LIN {X 0,Y 316.116,Z 363.716,A -85,B 0,C 180,E1 -15587.061,E2 -15587.061} C_VEL
LIN {X 0,Y 317.53,Z 353.599,A -85,B 0,C 180,E1 -15588.551,E2 -15588.551} C_VEL
LIN {X 0,Y 318.947,Z 342.978,A -85,B 0,C 180,E1 -15589.802,E2 -15589.802} C_VEL
LIN {X 0,Y 320.341,Z 331.099,A -85,B 0,C 180,E1 -15590.885,E2 -15590.885} C_VEL
LIN {X 0,Y 321.512,Z 318.732,A -85,B 0,C 180,E1 -15591.729,E2 -15591.729} C_VEL
LIN {X 0,Y 322.42,Z 306.003,A -85,B 0,C 180,E1 -15592.339,E2 -15592.339} C_VEL
LIN {X 0,Y 322.987,Z 292.578,A -85,B 0,C 180,E1 -15592.719,E2 -15592.719} C_VEL
LIN {X 0,Y 324.316,Z 230.091,A -85,B 0,C 180,E1 -15594.097,E2 -15594.097} C_VEL
LIN {X 0,Y 319.347,Z 202.293,A -85,B 0,C 180,E1 -15595.169,E2 -15595.169} C_VEL
LIN {X 0,Y 318.009,Z 197.372,A -85,B 0,C 180,E1 -15595.402,E2 -15595.402} C_VEL
LIN {X 0,Y 316.408,Z 192.985,A -85,B 0,C 180,E1 -15595.706,E2 -15595.706} C_VEL
LIN {X 0,Y 314.523,Z 183.518,A -85,B 0,C 180,E1 -15598.663,E2 -15598.663} C_VEL
LIN {X 0,Y 312.488,Z 174.615,A -85,B 0,C 180,E1 -15601.724,E2 -15601.724} C_VEL
LIN {X 0,Y 312.503,Z 174.545,A -85,B 0,C 180,E1 -15604.209,E2 -15604.209} C_VEL
LIN {X 0,Y 312.511,Z 174.539,A -85,B 0,C 180,E1 -15607.385,E2 -15607.385} C_VEL
LIN {X 0,Y 312.484,Z 174.559,A -85,B 0,C 180,E1 -15610.708,E2 -15610.708} C_VEL
LIN {X 0,Y 312.446,Z 174.564,A -85,B 0,C 180,E1 -15614.209,E2 -15614.209} C_VEL
LIN {X 0,Y 312.478,Z 174.558,A -85,B 0,C 180,E1 -15617.918,E2 -15617.918} C_VEL
LIN {X 0,Y 312.496,Z 174.545,A -85,B 0,C 180,E1 -15620.971,E2 -15620.971} C_VEL
LIN {X 0,Y 312.524,Z 174.52,A -85,B 0,C 180,E1 -15624.219,E2 -15624.219} C_VEL
LIN {X 0,Y 312.496,Z 174.56,A -85,B 0,C 180,E1 -15627.333,E2 -15627.333} C_VEL
LIN {X 0,Y 312.536,Z 174.547,A -85,B 0,C 180,E1 -15631.278,E2 -15631.278} C_VEL
LIN {X 0,Y 312.575,Z 174.542,A -85,B 0,C 180,E1 -15634.71,E2 -15634.71} C_VEL
LIN {X 0,Y 312.524,Z 174.557,A -85,B 0,C 180,E1 -15638.912,E2 -15638.912} C_VEL
LIN {X 0,Y 312.579,Z 174.534,A -85,B 0,C 180,E1 -15641.653,E2 -15641.653} C_VEL
LIN {X 0,Y 312.676,Z 174.535,A -85,B 0,C 180,E1 -15645.685,E2 -15645.685} C_VEL
LIN {X 0,Y 312.693,Z 174.524,A -85,B 0,C 180,E1 -15649.642,E2 -15649.642} C_VEL
LIN {X 0,Y 312.855,Z 174.515,A -85,B 0,C 180,E1 -15652.254,E2 -15652.254} C_VEL
LIN {X 0,Y 312.702,Z 174.515,A -85,B 0,C 180,E1 -15654.842,E2 -15654.842} C_VEL
LIN {X 0,Y 312.979,Z 174.501,A -85,B 0,C 180,E1 -15658.713,E2 -15658.713} C_VEL
LIN {X 0,Y 312.979,Z 174.486,A -85,B 0,C 180,E1 -15661.287,E2 -15661.287} C_VEL
LIN {X 0,Y 312.704,Z 174.531,A -85,B 0,C 180,E1 -15665.158,E2 -15665.158} C_VEL
LIN {X 0,Y 312.862,Z 174.506,A -85,B 0,C 180,E1 -15667.746,E2 -15667.746} C_VEL
LIN {X 0,Y 312.659,Z 174.534,A -85,B 0,C 180,E1 -15671.672,E2 -15671.672} C_VEL
LIN {X 0,Y 312.69,Z 174.521,A -85,B 0,C 180,E1 -15674.888,E2 -15674.888} C_VEL
LIN {X 0,Y 312.621,Z 174.542,A -85,B 0,C 180,E1 -15679.237,E2 -15679.237} C_VEL
LIN {X 0,Y 312.537,Z 174.544,A -85,B 0,C 180,E1 -15682.79,E2 -15682.79} C_VEL
LIN {X 0,Y 312.594,Z 174.546,A -85,B 0,C 180,E1 -15685.936,E2 -15685.936} C_VEL
LIN {X 0,Y 312.537,Z 174.551,A -85,B 0,C 180,E1 -15689.651,E2 -15689.651} C_VEL
LIN {X 0,Y 312.512,Z 174.525,A -85,B 0,C 180,E1 -15693.69,E2 -15693.69} C_VEL
LIN {X 0,Y 312.519,Z 174.539,A -85,B 0,C 180,E1 -15697.386,E2 -15697.386} C_VEL
LIN {X 0,Y 312.484,Z 174.556,A -85,B 0,C 180,E1 -15700.71,E2 -15700.71} C_VEL
LIN {X 0,Y 312.446,Z 174.538,A -85,B 0,C 180,E1 -15704.211,E2 -15704.211} C_VEL
LIN {X 0,Y 312.479,Z 174.555,A -85,B 0,C 180,E1 -15707.92,E2 -15707.92} C_VEL
LIN {X 0,Y 312.494,Z 174.538,A -85,B 0,C 180,E1 -15710.972,E2 -15710.972} C_VEL
LIN {X 0,Y 312.529,Z 174.544,A -85,B 0,C 180,E1 -15714.222,E2 -15714.222} C_VEL
LIN {X 0,Y 312.502,Z 174.56,A -85,B 0,C 180,E1 -15717.335,E2 -15717.335} C_VEL
LIN {X 0,Y 312.588,Z 174.751,A -85,B 0,C 180,E1 -15719.892,E2 -15719.892} C_VEL
LIN {X 0,Y 314.789,Z 184.623,A -85,B 0,C 180,E1 -15723.259,E2 -15723.259} C_VEL
LIN {X 0,Y 315.444,Z 187.959,A -85,B 0,C 180,E1 -15724.271,E2 -15724.271} C_VEL
LIN {X 0,Y 320.254,Z 200.27,A -85,B 0,C 180,E1 -15725.032,E2 -15725.032} C_VEL
LIN {X 0,Y 324.375,Z 221.605,A -85,B 0,C 180,E1 -15725.88,E2 -15725.88} C_VEL
LIN {X 0,Y 322.885,Z 294.83,A -85,B 0,C 180,E1 -15727.527,E2 -15727.527} C_VEL
LIN {X 0,Y 322.027,Z 308.231,A -85,B 0,C 180,E1 -15728.055,E2 -15728.055} C_VEL
LIN {X 0,Y 321.046,Z 321.006,A -85,B 0,C 180,E1 -15728.827,E2 -15728.827} C_VEL
LIN {X 0,Y 319.867,Z 332.351,A -85,B 0,C 180,E1 -15729.755,E2 -15729.755} C_VEL
LIN {X 0,Y 318.375,Z 344.014,A -85,B 0,C 180,E1 -15730.999,E2 -15730.999} C_VEL
LIN {X 0,Y 316.985,Z 354.593,A -85,B 0,C 180,E1 -15732.435,E2 -15732.435} C_VEL
LIN {X 0,Y 315.832,Z 363.045,A -85,B 0,C 180,E1 -15733.851,E2 -15733.851} C_VEL
LIN {X 0,Y 314.535,Z 370.933,A -85,B 0,C 180,E1 -15735.442,E2 -15735.442} C_VEL
LIN {X 0,Y 313.25,Z 378.643,A -85,B 0,C 180,E1 -15737.365,E2 -15737.365} C_VEL
LIN {X 0,Y 312.168,Z 385.722,A -85,B 0,C 180,E1 -15739.625,E2 -15739.625} C_VEL
LIN {X 0,Y 311.5,Z 390.438,A -85,B 0,C 180,E1 -15741.568,E2 -15741.568} C_VEL
LIN {X 0,Y 311.007,Z 394.632,A -85,B 0,C 180,E1 -15743.879,E2 -15743.879} C_VEL
LIN {X 0,Y 310.803,Z 397.316,A -85,B 0,C 180,E1 -15746.111,E2 -15746.111} C_VEL
LIN {X 0,Y 310.698,Z 398.314,A -85,B 0,C 180,E1 -15747.408,E2 -15747.408} C_VEL
LIN {X 0,Y 310.619,Z 399.162,A -85,B 0,C 180,E1 -15750.001,E2 -15750.001} C_VEL
LIN {X 0,Y 310.622,Z 398.969,A -85,B 0,C 180,E1 -15751.297,E2 -15751.297} C_VEL
LIN {X 0,Y 310.697,Z 398.381,A -85,B 0,C 180,E1 -15752.593,E2 -15752.593} C_VEL
LIN {X 0,Y 310.797,Z 397.408,A -85,B 0,C 180,E1 -15753.89,E2 -15753.89} C_VEL
LIN {X 0,Y 311.027,Z 394.734,A -85,B 0,C 180,E1 -15756.157,E2 -15756.157} C_VEL
LIN {X 0,Y 311.497,Z 390.68,A -85,B 0,C 180,E1 -15758.433,E2 -15758.433} C_VEL
LIN {X 0,Y 312.123,Z 386.029,A -85,B 0,C 180,E1 -15760.378,E2 -15760.378} C_VEL
LIN {X 0,Y 313.176,Z 379.019,A -85,B 0,C 180,E1 -15762.639,E2 -15762.639} C_VEL
LIN {X 0,Y 314.476,Z 371.424,A -85,B 0,C 180,E1 -15764.562,E2 -15764.562} C_VEL
LIN {X 0,Y 315.716,Z 363.643,A -85,B 0,C 180,E1 -15766.156,E2 -15766.156} C_VEL
LIN {X 0,Y 317.118,Z 353.168,A -85,B 0,C 180,E1 -15767.894,E2 -15767.894} C_VEL
LIN {X 0,Y 318.634,Z 342.298,A -85,B 0,C 180,E1 -15769.32,E2 -15769.32} C_VEL
LIN {X 0,Y 319.963,Z 331.792,A -85,B 0,C 180,E1 -15770.408,E2 -15770.408} C_VEL
LIN {X 0,Y 321.208,Z 319.141,A -85,B 0,C 180,E1 -15771.415,E2 -15771.415} C_VEL
LIN {X 0,Y 322.223,Z 306.471,A -85,B 0,C 180,E1 -15772.143,E2 -15772.143} C_VEL
LIN {X 0,Y 322.942,Z 294.403,A -85,B 0,C 180,E1 -15772.597,E2 -15772.597} C_VEL
LIN {X 0,Y 324.453,Z 221.803,A -85,B 0,C 180,E1 -15774.224,E2 -15774.224} C_VEL
LIN {X 0,Y 320.487,Z 200.978,A -85,B 0,C 180,E1 -15775.047,E2 -15775.047} C_VEL
LIN {X 0,Y 315.485,Z 188.183,A -85,B 0,C 180,E1 -15775.822,E2 -15775.822} C_VEL
LIN {X 0,Y 314.974,Z 185.72,A -85,B 0,C 180,E1 -15776.504,E2 -15776.504} C_VEL
LIN {X 0,Y 312.776,Z 175.319,A -85,B 0,C 180,E1 -15779.997,E2 -15779.997} C_VEL
LIN {X 0,Y 312.588,Z 174.569,A -85,B 0,C 180,E1 -15780.389,E2 -15780.389} C_VEL
LIN {X 0,Y 312.507,Z 174.544,A -85,B 0,C 180,E1 -15784.21,E2 -15784.21} C_VEL
LIN {X 0,Y 312.521,Z 174.552,A -85,B 0,C 180,E1 -15787.089,E2 -15787.089} C_VEL
LIN {X 0,Y 311.895,Z 174.641,A -85,B 0,C 180,E1 -15788.164,E2 -15788.164} C_VEL
LIN {X 0,Y 309.062,Z 174.996,A -85,B 0,C 180,E1 -15789.915,E2 -15789.915} C_VEL
LIN {X 0,Y 306.618,Z 175.294,A -85,B 0,C 180,E1 -15791.335,E2 -15791.335} C_VEL
LIN {X 0,Y 305.541,Z 175.424,A -85,B 0,C 180,E1 -15792.434,E2 -15792.434} C_VEL
LIN {X 0,Y 305.439,Z 175.436,A -85,B 0,C 180,E1 -15792.807,E2 -15792.807} C_VEL
LIN {X 0,Y 305.454,Z 175.406,A -85,B 0,C 180,E1 -15797.414,E2 -15797.414} C_VEL
LIN {X 0,Y 305.475,Z 175.43,A -85,B 0,C 180,E1 -15801.597,E2 -15801.597} C_VEL
LIN {X 0,Y 305.46,Z 175.388,A -85,B 0,C 180,E1 -15804.886,E2 -15804.886} C_VEL
LIN {X 0,Y 305.45,Z 175.432,A -85,B 0,C 180,E1 -15808.355,E2 -15808.355} C_VEL
LIN {X 0,Y 305.518,Z 175.425,A -85,B 0,C 180,E1 -15811.113,E2 -15811.113} C_VEL
LIN {X 0,Y 305.568,Z 175.42,A -85,B 0,C 180,E1 -15814.087,E2 -15814.087} C_VEL
LIN {X 0,Y 305.477,Z 175.42,A -85,B 0,C 180,E1 -15818.401,E2 -15818.401} C_VEL
LIN {X 0,Y 305.576,Z 175.421,A -85,B 0,C 180,E1 -15821.217,E2 -15821.217} C_VEL
LIN {X 0,Y 305.645,Z 175.399,A -85,B 0,C 180,E1 -15825.349,E2 -15825.349} C_VEL
LIN {X 0,Y 305.634,Z 175.403,A -85,B 0,C 180,E1 -15829.399,E2 -15829.399} C_VEL
LIN {X 0,Y 305.809,Z 175.38,A -85,B 0,C 180,E1 -15832.074,E2 -15832.074} C_VEL
LIN {X 0,Y 305.681,Z 175.405,A -85,B 0,C 180,E1 -15834.723,E2 -15834.723} C_VEL
LIN {X 0,Y 305.952,Z 175.362,A -85,B 0,C 180,E1 -15838.684,E2 -15838.684} C_VEL
LIN {X 0,Y 305.95,Z 175.376,A -85,B 0,C 180,E1 -15841.316,E2 -15841.316} C_VEL
LIN {X 0,Y 305.675,Z 175.391,A -85,B 0,C 180,E1 -15845.277,E2 -15845.277} C_VEL
LIN {X 0,Y 305.767,Z 175.397,A -85,B 0,C 180,E1 -15847.927,E2 -15847.927} C_VEL
LIN {X 0,Y 305.593,Z 175.404,A -85,B 0,C 180,E1 -15851.945,E2 -15851.945} C_VEL
LIN {X 0,Y 305.605,Z 175.418,A -85,B 0,C 180,E1 -15855.014,E2 -15855.014} C_VEL
LIN {X 0,Y 305.543,Z 175.419,A -85,B 0,C 180,E1 -15859.429,E2 -15859.429} C_VEL
LIN {X 0,Y 305.483,Z 175.422,A -85,B 0,C 180,E1 -15863.04,E2 -15863.04} C_VEL
LIN {X 0,Y 305.528,Z 175.426,A -85,B 0,C 180,E1 -15866.221,E2 -15866.221} C_VEL
LIN {X 0,Y 305.485,Z 175.422,A -85,B 0,C 180,E1 -15869.047,E2 -15869.047} C_VEL
LIN {X 0,Y 305.439,Z 175.438,A -85,B 0,C 180,E1 -15871.953,E2 -15871.953} C_VEL
LIN {X 0,Y 305.459,Z 175.406,A -85,B 0,C 180,E1 -15875.114,E2 -15875.114} C_VEL
LIN {X 0,Y 305.447,Z 175.418,A -85,B 0,C 180,E1 -15878.529,E2 -15878.529} C_VEL
LIN {X 0,Y 305.453,Z 175.428,A -85,B 0,C 180,E1 -15882.586,E2 -15882.586} C_VEL
LIN {X 0,Y 305.424,Z 175.436,A -85,B 0,C 180,E1 -15886.345,E2 -15886.345} C_VEL
LIN {X 0,Y 305.456,Z 175.427,A -85,B 0,C 180,E1 -15889.892,E2 -15889.892} C_VEL
LIN {X 0,Y 305.478,Z 175.432,A -85,B 0,C 180,E1 -15893.633,E2 -15893.633} C_VEL
LIN {X 0,Y 305.463,Z 175.515,A -85,B 0,C 180,E1 -15897.759,E2 -15897.759} C_VEL
LIN {X 0,Y 307.544,Z 184.711,A -85,B 0,C 180,E1 -15900.991,E2 -15900.991} C_VEL
LIN {X 0,Y 309.22,Z 192.944,A -85,B 0,C 180,E1 -15903.631,E2 -15903.631} C_VEL
LIN {X 0,Y 312.213,Z 200.76,A -85,B 0,C 180,E1 -15904.151,E2 -15904.151} C_VEL
LIN {X 0,Y 314.705,Z 212.364,A -85,B 0,C 180,E1 -15904.657,E2 -15904.657} C_VEL
LIN {X 0,Y 317.835,Z 230.736,A -85,B 0,C 180,E1 -15905.371,E2 -15905.371} C_VEL
LIN {X 0,Y 316.219,Z 300.948,A -85,B 0,C 180,E1 -15906.982,E2 -15906.982} C_VEL
LIN {X 0,Y 315.294,Z 314.872,A -85,B 0,C 180,E1 -15907.56,E2 -15907.56} C_VEL
LIN {X 0,Y 314.138,Z 327.319,A -85,B 0,C 180,E1 -15908.337,E2 -15908.337} C_VEL
LIN {X 0,Y 312.931,Z 338.417,A -85,B 0,C 180,E1 -15909.285,E2 -15909.285} C_VEL
LIN {X 0,Y 311.387,Z 349.974,A -85,B 0,C 180,E1 -15910.555,E2 -15910.555} C_VEL
LIN {X 0,Y 309.787,Z 360.7,A -85,B 0,C 180,E1 -15912.046,E2 -15912.046} C_VEL
LIN {X 0,Y 308.277,Z 370.627,A -85,B 0,C 180,E1 -15913.798,E2 -15913.798} C_VEL
LIN {X 0,Y 306.817,Z 379.458,A -85,B 0,C 180,E1 -15915.745,E2 -15915.745} C_VEL
LIN {X 0,Y 305.632,Z 386.621,A -85,B 0,C 180,E1 -15917.719,E2 -15917.719} C_VEL
LIN {X 0,Y 304.624,Z 393.142,A -85,B 0,C 180,E1 -15920.035,E2 -15920.035} C_VEL
LIN {X 0,Y 304.056,Z 397.456,A -85,B 0,C 180,E1 -15922.028,E2 -15922.028} C_VEL
LIN {X 0,Y 303.73,Z 401.017,A -85,B 0,C 180,E1 -15924.256,E2 -15924.256} C_VEL
LIN {X 0,Y 303.612,Z 402.976,A -85,B 0,C 180,E1 -15926.017,E2 -15926.017} C_VEL
LIN {X 0,Y 303.585,Z 403.966,A -85,B 0,C 180,E1 -15927.346,E2 -15927.346} C_VEL
LIN {X 0,Y 303.528,Z 404.568,A -85,B 0,C 180,E1 -15928.673,E2 -15928.673} C_VEL
LIN {X 0,Y 303.533,Z 404.78,A -85,B 0,C 180,E1 -15929.999,E2 -15929.999} C_VEL
LIN {X 0,Y 303.585,Z 403.954,A -85,B 0,C 180,E1 -15932.653,E2 -15932.653} C_VEL
LIN {X 0,Y 303.612,Z 402.961,A -85,B 0,C 180,E1 -15933.981,E2 -15933.981} C_VEL
LIN {X 0,Y 303.782,Z 400.858,A -85,B 0,C 180,E1 -15935.841,E2 -15935.841} C_VEL
LIN {X 0,Y 304.094,Z 397.415,A -85,B 0,C 180,E1 -15937.97,E2 -15937.97} C_VEL
LIN {X 0,Y 304.623,Z 393.087,A -85,B 0,C 180,E1 -15939.963,E2 -15939.963} C_VEL
LIN {X 0,Y 305.46,Z 387.573,A -85,B 0,C 180,E1 -15941.95,E2 -15941.95} C_VEL
LIN {X 0,Y 306.61,Z 380.689,A -85,B 0,C 180,E1 -15943.926,E2 -15943.926} C_VEL
LIN {X 0,Y 308.023,Z 372.072,A -85,B 0,C 180,E1 -15945.889,E2 -15945.889} C_VEL
LIN {X 0,Y 309.342,Z 363.431,A -85,B 0,C 180,E1 -15947.484,E2 -15947.484} C_VEL
LIN {X 0,Y 310.813,Z 353.531,A -85,B 0,C 180,E1 -15948.967,E2 -15948.967} C_VEL
LIN {X 0,Y 312.267,Z 342.909,A -85,B 0,C 180,E1 -15950.244,E2 -15950.244} C_VEL
LIN {X 0,Y 313.728,Z 331.028,A -85,B 0,C 180,E1 -15951.346,E2 -15951.346} C_VEL
LIN {X 0,Y 314.943,Z 318.659,A -85,B 0,C 180,E1 -15952.206,E2 -15952.206} C_VEL
LIN {X 0,Y 315.884,Z 305.927,A -85,B 0,C 180,E1 -15952.827,E2 -15952.827} C_VEL
LIN {X 0,Y 316.461,Z 292.492,A -85,B 0,C 180,E1 -15953.215,E2 -15953.215} C_VEL
LIN {X 0,Y 317.799,Z 230.975,A -85,B 0,C 180,E1 -15954.6,E2 -15954.6} C_VEL
LIN {X 0,Y 313.092,Z 204.209,A -85,B 0,C 180,E1 -15955.658,E2 -15955.658} C_VEL
LIN {X 0,Y 311.692,Z 199.331,A -85,B 0,C 180,E1 -15955.903,E2 -15955.903} C_VEL
LIN {X 0,Y 309.197,Z 193.025,A -85,B 0,C 180,E1 -15956.332,E2 -15956.332} C_VEL
LIN {X 0,Y 307.519,Z 184.646,A -85,B 0,C 180,E1 -15959.001,E2 -15959.001} C_VEL
LIN {X 0,Y 305.472,Z 175.62,A -85,B 0,C 180,E1 -15962.142,E2 -15962.142} C_VEL
LIN {X 0,Y 305.458,Z 175.43,A -85,B 0,C 180,E1 -15965.112,E2 -15965.112} C_VEL
LIN {X 0,Y 305.422,Z 175.415,A -85,B 0,C 180,E1 -15968.522,E2 -15968.522} C_VEL
LIN {X 0,Y 305.435,Z 175.437,A -85,B 0,C 180,E1 -15971.856,E2 -15971.856} C_VEL
LIN {X 0,Y 305.394,Z 175.441,A -85,B 0,C 180,E1 -15975.51,E2 -15975.51} C_VEL
LIN {X 0,Y 305.434,Z 175.435,A -85,B 0,C 180,E1 -15978.142,E2 -15978.142} C_VEL
LIN {X 0,Y 305.469,Z 175.41,A -85,B 0,C 180,E1 -15981.596,E2 -15981.596} C_VEL
LIN {X 0,Y 305.455,Z 175.408,A -85,B 0,C 180,E1 -15984.886,E2 -15984.886} C_VEL
LIN {X 0,Y 305.441,Z 175.438,A -85,B 0,C 180,E1 -15988.355,E2 -15988.355} C_VEL
LIN {X 0,Y 305.505,Z 175.421,A -85,B 0,C 180,E1 -15991.112,E2 -15991.112} C_VEL
LIN {X 0,Y 305.562,Z 175.421,A -85,B 0,C 180,E1 -15994.087,E2 -15994.087} C_VEL
LIN {X 0,Y 305.47,Z 175.433,A -85,B 0,C 180,E1 -15998.401,E2 -15998.401} C_VEL
LIN {X 0,Y 305.539,Z 175.412,A -85,B 0,C 180,E1 -16001.214,E2 -16001.214} C_VEL
LIN {X 0,Y 305.616,Z 175.415,A -85,B 0,C 180,E1 -16005.347,E2 -16005.347} C_VEL
LIN {X 0,Y 305.629,Z 175.402,A -85,B 0,C 180,E1 -16009.399,E2 -16009.399} C_VEL
LIN {X 0,Y 305.798,Z 175.393,A -85,B 0,C 180,E1 -16012.074,E2 -16012.074} C_VEL
LIN {X 0,Y 305.674,Z 175.391,A -85,B 0,C 180,E1 -16014.723,E2 -16014.723} C_VEL
LIN {X 0,Y 305.946,Z 175.377,A -85,B 0,C 180,E1 -16018.684,E2 -16018.684} C_VEL
LIN {X 0,Y 305.946,Z 175.362,A -85,B 0,C 180,E1 -16021.316,E2 -16021.316} C_VEL
LIN {X 0,Y 305.84,Z 175.385,A -85,B 0,C 180,E1 -16026.598,E2 -16026.598} C_VEL
LIN {X 0,Y 305.726,Z 175.381,A -85,B 0,C 180,E1 -16029.26,E2 -16029.26} C_VEL
LIN {X 0,Y 305.579,Z 175.417,A -85,B 0,C 180,E1 -16033.297,E2 -16033.297} C_VEL
LIN {X 0,Y 305.584,Z 175.403,A -85,B 0,C 180,E1 -16036.021,E2 -16036.021} C_VEL
LIN {X 0,Y 305.568,Z 175.421,A -85,B 0,C 180,E1 -16039.445,E2 -16039.445} C_VEL
LIN {X 0,Y 305.482,Z 175.425,A -85,B 0,C 180,E1 -16043.042,E2 -16043.042} C_VEL
LIN {X 0,Y 305.524,Z 175.423,A -85,B 0,C 180,E1 -16046.222,E2 -16046.222} C_VEL
LIN {X 0,Y 305.488,Z 175.428,A -85,B 0,C 180,E1 -16049.051,E2 -16049.051} C_VEL
LIN {X 0,Y 305.437,Z 175.431,A -85,B 0,C 180,E1 -16051.953,E2 -16051.953} C_VEL
LIN {X 0,Y 305.455,Z 175.39,A -85,B 0,C 180,E1 -16055.114,E2 -16055.114} C_VEL
LIN {X 0,Y 305.443,Z 175.434,A -85,B 0,C 180,E1 -16058.53,E2 -16058.53} C_VEL
LIN {X 0,Y 305.449,Z 175.409,A -85,B 0,C 180,E1 -16062.587,E2 -16062.587} C_VEL
LIN {X 0,Y 305.421,Z 175.441,A -85,B 0,C 180,E1 -16066.346,E2 -16066.346} C_VEL
LIN {X 0,Y 305.454,Z 175.41,A -85,B 0,C 180,E1 -16069.894,E2 -16069.894} C_VEL
LIN {X 0,Y 305.477,Z 175.429,A -85,B 0,C 180,E1 -16073.633,E2 -16073.633} C_VEL
LIN {X 0,Y 305.462,Z 175.428,A -85,B 0,C 180,E1 -16076.485,E2 -16076.485} C_VEL
LIN {X 0,Y 305.514,Z 175.51,A -85,B 0,C 180,E1 -16079.311,E2 -16079.311} C_VEL
LIN {X 0,Y 307.81,Z 185.73,A -85,B 0,C 180,E1 -16082.931,E2 -16082.931} C_VEL
LIN {X 0,Y 308.278,Z 188.103,A -85,B 0,C 180,E1 -16083.636,E2 -16083.636} C_VEL
LIN {X 0,Y 314.35,Z 203.461,A -85,B 0,C 180,E1 -16084.607,E2 -16084.607} C_VEL
LIN {X 0,Y 317.972,Z 223.57,A -85,B 0,C 180,E1 -16085.408,E2 -16085.408} C_VEL
LIN {X 0,Y 316.28,Z 296.069,A -85,B 0,C 180,E1 -16087.074,E2 -16087.074} C_VEL
LIN {X 0,Y 315.368,Z 309.828,A -85,B 0,C 180,E1 -16087.653,E2 -16087.653} C_VEL
LIN {X 0,Y 314.332,Z 322.174,A -85,B 0,C 180,E1 -16088.438,E2 -16088.438} C_VEL
LIN {X 0,Y 313.007,Z 334.008,A -85,B 0,C 180,E1 -16089.463,E2 -16089.463} C_VEL
LIN {X 0,Y 311.505,Z 345.373,A -85,B 0,C 180,E1 -16090.735,E2 -16090.735} C_VEL
LIN {X 0,Y 310.107,Z 355.391,A -85,B 0,C 180,E1 -16092.149,E2 -16092.149} C_VEL
LIN {X 0,Y 308.726,Z 364.809,A -85,B 0,C 180,E1 -16093.809,E2 -16093.809} C_VEL
LIN {X 0,Y 307.129,Z 373.744,A -85,B 0,C 180,E1 -16095.761,E2 -16095.761} C_VEL
LIN {X 0,Y 305.971,Z 380.937,A -85,B 0,C 180,E1 -16097.734,E2 -16097.734} C_VEL
LIN {X 0,Y 305.159,Z 385.789,A -85,B 0,C 180,E1 -16099.384,E2 -16099.384} C_VEL
LIN {X 0,Y 304.467,Z 390.504,A -85,B 0,C 180,E1 -16101.372,E2 -16101.372} C_VEL
LIN {X 0,Y 304.007,Z 394.113,A -85,B 0,C 180,E1 -16103.363,E2 -16103.363} C_VEL
LIN {X 0,Y 303.819,Z 395.978,A -85,B 0,C 180,E1 -16104.692,E2 -16104.692} C_VEL
LIN {X 0,Y 303.72,Z 397.381,A -85,B 0,C 180,E1 -16106.02,E2 -16106.02} C_VEL
LIN {X 0,Y 303.626,Z 398.38,A -85,B 0,C 180,E1 -16107.347,E2 -16107.347} C_VEL
LIN {X 0,Y 303.535,Z 399.226,A -85,B 0,C 180,E1 -16110.001,E2 -16110.001} C_VEL
LIN {X 0,Y 303.541,Z 399.034,A -85,B 0,C 180,E1 -16111.327,E2 -16111.327} C_VEL
LIN {X 0,Y 303.625,Z 398.445,A -85,B 0,C 180,E1 -16112.654,E2 -16112.654} C_VEL
LIN {X 0,Y 303.714,Z 397.473,A -85,B 0,C 180,E1 -16113.981,E2 -16113.981} C_VEL
LIN {X 0,Y 303.936,Z 395.045,A -85,B 0,C 180,E1 -16116.116,E2 -16116.116} C_VEL
LIN {X 0,Y 304.299,Z 392.029,A -85,B 0,C 180,E1 -16117.966,E2 -16117.966} C_VEL
LIN {X 0,Y 304.861,Z 387.759,A -85,B 0,C 180,E1 -16119.957,E2 -16119.957} C_VEL
LIN {X 0,Y 305.937,Z 381.296,A -85,B 0,C 180,E1 -16122.269,E2 -16122.269} C_VEL
LIN {X 0,Y 307.079,Z 374.196,A -85,B 0,C 180,E1 -16124.243,E2 -16124.243} C_VEL
LIN {X 0,Y 308.644,Z 365.351,A -85,B 0,C 180,E1 -16126.197,E2 -16126.197} C_VEL
LIN {X 0,Y 309.988,Z 355.877,A -85,B 0,C 180,E1 -16127.893,E2 -16127.893} C_VEL
LIN {X 0,Y 311.388,Z 346.231,A -85,B 0,C 180,E1 -16129.274,E2 -16129.274} C_VEL
LIN {X 0,Y 312.943,Z 335.054,A -85,B 0,C 180,E1 -16130.543,E2 -16130.543} C_VEL
LIN {X 0,Y 314.342,Z 322.512,A -85,B 0,C 180,E1 -16131.648,E2 -16131.648} C_VEL
LIN {X 0,Y 315.448,Z 309.573,A -85,B 0,C 180,E1 -16132.472,E2 -16132.472} C_VEL
LIN {X 0,Y 316.29,Z 296.811,A -85,B 0,C 180,E1 -16133.013,E2 -16133.013} C_VEL
LIN {X 0,Y 317.119,Z 265.233,A -85,B 0,C 180,E1 -16133.765,E2 -16133.765} C_VEL
LIN {X 0,Y 317.973,Z 222.627,A -85,B 0,C 180,E1 -16134.731,E2 -16134.731} C_VEL
LIN {X 0,Y 314.219,Z 203.145,A -85,B 0,C 180,E1 -16135.53,E2 -16135.53} C_VEL
LIN {X 0,Y 308.264,Z 188.057,A -85,B 0,C 180,E1 -16136.491,E2 -16136.491} C_VEL
LIN {X 0,Y 306.44,Z 179.396,A -85,B 0,C 180,E1 -16139.366,E2 -16139.366} C_VEL
LIN {X 0,Y 305.509,Z 175.49,A -85,B 0,C 180,E1 -16140.835,E2 -16140.835} C_VEL
LIN {X 0,Y 305.463,Z 175.418,A -85,B 0,C 180,E1 -16145.113,E2 -16145.113} C_VEL
LIN {X 0,Y 305.449,Z 175.424,A -85,B 0,C 180,E1 -16148.528,E2 -16148.528} C_VEL
LIN {X 0,Y 305.454,Z 175.435,A -85,B 0,C 180,E1 -16152.585,E2 -16152.585} C_VEL
LIN {X 0,Y 305.439,Z 175.436,A -85,B 0,C 180,E1 -16152.807,E2 -16152.807} C_VEL
LIN {X 0,Y 304.725,Z 175.526,A -85,B 0,C 180,E1 -16153.907,E2 -16153.907} C_VEL
LIN {X 0,Y 301.828,Z 175.865,A -85,B 0,C 180,E1 -16155.696,E2 -16155.696} C_VEL
LIN {X 0,Y 299.424,Z 176.157,A -85,B 0,C 180,E1 -16157.148,E2 -16157.148} C_VEL
LIN {X 0,Y 298.436,Z 176.289,A -85,B 0,C 180,E1 -16158.273,E2 -16158.273} C_VEL
LIN {X 0,Y 298.378,Z 176.302,A -85,B 0,C 180,E1 -16158.654,E2 -16158.654} C_VEL
LIN {X 0,Y 298.412,Z 176.302,A -85,B 0,C 180,E1 -16162.241,E2 -16162.241} C_VEL
LIN {X 0,Y 298.406,Z 176.268,A -85,B 0,C 180,E1 -16165.581,E2 -16165.581} C_VEL
LIN {X 0,Y 298.393,Z 176.314,A -85,B 0,C 180,E1 -16168.791,E2 -16168.791} C_VEL
LIN {X 0,Y 298.46,Z 176.296,A -85,B 0,C 180,E1 -16171.904,E2 -16171.904} C_VEL
LIN {X 0,Y 298.481,Z 176.304,A -85,B 0,C 180,E1 -16174.923,E2 -16174.923} C_VEL
LIN {X 0,Y 298.433,Z 176.302,A -85,B 0,C 180,E1 -16179.314,E2 -16179.314} C_VEL
LIN {X 0,Y 298.531,Z 176.294,A -85,B 0,C 180,E1 -16182.179,E2 -16182.179} C_VEL
LIN {X 0,Y 298.59,Z 176.276,A -85,B 0,C 180,E1 -16184.994,E2 -16184.994} C_VEL
LIN {X 0,Y 298.59,Z 176.284,A -85,B 0,C 180,E1 -16189.146,E2 -16189.146} C_VEL
LIN {X 0,Y 298.755,Z 176.256,A -85,B 0,C 180,E1 -16191.886,E2 -16191.886} C_VEL
LIN {X 0,Y 298.652,Z 176.281,A -85,B 0,C 180,E1 -16194.599,E2 -16194.599} C_VEL
LIN {X 0,Y 298.918,Z 176.238,A -85,B 0,C 180,E1 -16198.653,E2 -16198.653} C_VEL
LIN {X 0,Y 298.917,Z 176.252,A -85,B 0,C 180,E1 -16201.347,E2 -16201.347} C_VEL
LIN {X 0,Y 298.77,Z 176.263,A -85,B 0,C 180,E1 -16206.754,E2 -16206.754} C_VEL
LIN {X 0,Y 298.621,Z 176.281,A -85,B 0,C 180,E1 -16209.482,E2 -16209.482} C_VEL
LIN {X 0,Y 298.54,Z 176.295,A -85,B 0,C 180,E1 -16213.616,E2 -16213.616} C_VEL
LIN {X 0,Y 298.483,Z 176.299,A -85,B 0,C 180,E1 -16216.412,E2 -16216.412} C_VEL
LIN {X 0,Y 298.483,Z 176.301,A -85,B 0,C 180,E1 -16219.641,E2 -16219.641} C_VEL
LIN {X 0,Y 298.426,Z 176.297,A -85,B 0,C 180,E1 -16223.6,E2 -16223.6} C_VEL
LIN {X 0,Y 298.484,Z 176.304,A -85,B 0,C 180,E1 -16226.575,E2 -16226.575} C_VEL
LIN {X 0,Y 298.414,Z 176.303,A -85,B 0,C 180,E1 -16229.642,E2 -16229.642} C_VEL
LIN {X 0,Y 298.392,Z 176.315,A -85,B 0,C 180,E1 -16232.801,E2 -16232.801} C_VEL
LIN {X 0,Y 298.444,Z 176.267,A -85,B 0,C 180,E1 -16236.808,E2 -16236.808} C_VEL
LIN {X 0,Y 298.385,Z 176.317,A -85,B 0,C 180,E1 -16241.088,E2 -16241.088} C_VEL
LIN {X 0,Y 298.398,Z 176.305,A -85,B 0,C 180,E1 -16243.104,E2 -16243.104} C_VEL
LIN {X 0,Y 298.402,Z 176.307,A -85,B 0,C 180,E1 -16246.921,E2 -16246.921} C_VEL
LIN {X 0,Y 298.389,Z 176.293,A -85,B 0,C 180,E1 -16251.01,E2 -16251.01} C_VEL
LIN {X 0,Y 298.417,Z 176.315,A -85,B 0,C 180,E1 -16253.93,E2 -16253.93} C_VEL
LIN {X 0,Y 298.463,Z 176.375,A -85,B 0,C 180,E1 -16257.208,E2 -16257.208} C_VEL
LIN {X 0,Y 300.544,Z 185.697,A -85,B 0,C 180,E1 -16260.589,E2 -16260.589} C_VEL
LIN {X 0,Y 302.053,Z 192.974,A -85,B 0,C 180,E1 -16262.968,E2 -16262.968} C_VEL
LIN {X 0,Y 306.642,Z 205.052,A -85,B 0,C 180,E1 -16263.756,E2 -16263.756} C_VEL
LIN {X 0,Y 311.027,Z 229.598,A -85,B 0,C 180,E1 -16264.768,E2 -16264.768} C_VEL
LIN {X 0,Y 311.41,Z 233.755,A -85,B 0,C 180,E1 -16264.905,E2 -16264.905} C_VEL
LIN {X 0,Y 309.706,Z 300.897,A -85,B 0,C 180,E1 -16266.469,E2 -16266.469} C_VEL
LIN {X 0,Y 308.76,Z 314.816,A -85,B 0,C 180,E1 -16267.058,E2 -16267.058} C_VEL
LIN {X 0,Y 307.537,Z 327.26,A -85,B 0,C 180,E1 -16267.848,E2 -16267.848} C_VEL
LIN {X 0,Y 306.287,Z 338.356,A -85,B 0,C 180,E1 -16268.814,E2 -16268.814} C_VEL
LIN {X 0,Y 304.698,Z 349.913,A -85,B 0,C 180,E1 -16270.11,E2 -16270.11} C_VEL
LIN {X 0,Y 303.06,Z 360.317,A -85,B 0,C 180,E1 -16271.581,E2 -16271.581} C_VEL
LIN {X 0,Y 301.668,Z 369.306,A -85,B 0,C 180,E1 -16273.166,E2 -16273.166} C_VEL
LIN {X 0,Y 300.199,Z 378.04,A -85,B 0,C 180,E1 -16275.077,E2 -16275.077} C_VEL
LIN {X 0,Y 298.837,Z 385.445,A -85,B 0,C 180,E1 -16277.09,E2 -16277.09} C_VEL
LIN {X 0,Y 297.864,Z 391.391,A -85,B 0,C 180,E1 -16279.119,E2 -16279.119} C_VEL
LIN {X 0,Y 297.199,Z 396.088,A -85,B 0,C 180,E1 -16281.158,E2 -16281.158} C_VEL
LIN {X 0,Y 296.762,Z 399.675,A -85,B 0,C 180,E1 -16283.199,E2 -16283.199} C_VEL
LIN {X 0,Y 296.601,Z 401.525,A -85,B 0,C 180,E1 -16284.561,E2 -16284.561} C_VEL
LIN {X 0,Y 296.516,Z 402.911,A -85,B 0,C 180,E1 -16285.922,E2 -16285.922} C_VEL
LIN {X 0,Y 296.491,Z 403.901,A -85,B 0,C 180,E1 -16287.282,E2 -16287.282} C_VEL
LIN {X 0,Y 296.45,Z 404.504,A -85,B 0,C 180,E1 -16288.641,E2 -16288.641} C_VEL
LIN {X 0,Y 296.451,Z 404.716,A -85,B 0,C 180,E1 -16289.999,E2 -16289.999} C_VEL
LIN {X 0,Y 296.45,Z 404.496,A -85,B 0,C 180,E1 -16291.358,E2 -16291.358} C_VEL
LIN {X 0,Y 296.491,Z 403.889,A -85,B 0,C 180,E1 -16292.717,E2 -16292.717} C_VEL
LIN {X 0,Y 296.64,Z 401.501,A -85,B 0,C 180,E1 -16295.437,E2 -16295.437} C_VEL
LIN {X 0,Y 296.897,Z 398.573,A -85,B 0,C 180,E1 -16297.48,E2 -16297.48} C_VEL
LIN {X 0,Y 297.384,Z 394.61,A -85,B 0,C 180,E1 -16299.521,E2 -16299.521} C_VEL
LIN {X 0,Y 298.356,Z 388.515,A -85,B 0,C 180,E1 -16301.894,E2 -16301.894} C_VEL
LIN {X 0,Y 299.465,Z 381.855,A -85,B 0,C 180,E1 -16303.918,E2 -16303.918} C_VEL
LIN {X 0,Y 300.938,Z 373.592,A -85,B 0,C 180,E1 -16305.926,E2 -16305.926} C_VEL
LIN {X 0,Y 302.285,Z 365.114,A -85,B 0,C 180,E1 -16307.591,E2 -16307.591} C_VEL
LIN {X 0,Y 303.713,Z 355.811,A -85,B 0,C 180,E1 -16309.077,E2 -16309.077} C_VEL
LIN {X 0,Y 305.398,Z 344.267,A -85,B 0,C 180,E1 -16310.544,E2 -16310.544} C_VEL
LIN {X 0,Y 306.909,Z 332.892,A -85,B 0,C 180,E1 -16311.668,E2 -16311.668} C_VEL
LIN {X 0,Y 308.171,Z 321.188,A -85,B 0,C 180,E1 -16312.544,E2 -16312.544} C_VEL
LIN {X 0,Y 309.226,Z 307.689,A -85,B 0,C 180,E1 -16313.258,E2 -16313.258} C_VEL
LIN {X 0,Y 309.908,Z 294.195,A -85,B 0,C 180,E1 -16313.691,E2 -16313.691} C_VEL
LIN {X 0,Y 311.288,Z 231.479,A -85,B 0,C 180,E1 -16315.135,E2 -16315.135} C_VEL
LIN {X 0,Y 306.724,Z 205.539,A -85,B 0,C 180,E1 -16316.195,E2 -16316.195} C_VEL
LIN {X 0,Y 304.353,Z 198.944,A -85,B 0,C 180,E1 -16316.584,E2 -16316.584} C_VEL
LIN {X 0,Y 302.015,Z 193.032,A -85,B 0,C 180,E1 -16316.998,E2 -16316.998} C_VEL
LIN {X 0,Y 301.27,Z 189.184,A -85,B 0,C 180,E1 -16318.188,E2 -16318.188} C_VEL
LIN {X 0,Y 299.079,Z 179.364,A -85,B 0,C 180,E1 -16321.606,E2 -16321.606} C_VEL
LIN {X 0,Y 298.425,Z 176.335,A -85,B 0,C 180,E1 -16322.795,E2 -16322.795} C_VEL
LIN {X 0,Y 298.438,Z 176.299,A -85,B 0,C 180,E1 -16326.805,E2 -16326.805} C_VEL
LIN {X 0,Y 298.382,Z 176.319,A -85,B 0,C 180,E1 -16331.086,E2 -16331.086} C_VEL
LIN {X 0,Y 298.394,Z 176.309,A -85,B 0,C 180,E1 -16333.102,E2 -16333.102} C_VEL
LIN {X 0,Y 298.397,Z 176.305,A -85,B 0,C 180,E1 -16336.92,E2 -16336.92} C_VEL
LIN {X 0,Y 298.397,Z 176.299,A -85,B 0,C 180,E1 -16341.005,E2 -16341.005} C_VEL
LIN {X 0,Y 298.411,Z 176.273,A -85,B 0,C 180,E1 -16343.929,E2 -16343.929} C_VEL
LIN {X 0,Y 298.386,Z 176.316,A -85,B 0,C 180,E1 -16347.983,E2 -16347.983} C_VEL
LIN {X 0,Y 298.45,Z 176.305,A -85,B 0,C 180,E1 -16351.903,E2 -16351.903} C_VEL
LIN {X 0,Y 298.475,Z 176.296,A -85,B 0,C 180,E1 -16354.923,E2 -16354.923} C_VEL
LIN {X 0,Y 298.423,Z 176.311,A -85,B 0,C 180,E1 -16359.313,E2 -16359.313} C_VEL
LIN {X 0,Y 298.496,Z 176.286,A -85,B 0,C 180,E1 -16362.177,E2 -16362.177} C_VEL
LIN {X 0,Y 298.577,Z 176.294,A -85,B 0,C 180,E1 -16364.994,E2 -16364.994} C_VEL
LIN {X 0,Y 298.585,Z 176.277,A -85,B 0,C 180,E1 -16369.146,E2 -16369.146} C_VEL
LIN {X 0,Y 298.744,Z 176.271,A -85,B 0,C 180,E1 -16371.886,E2 -16371.886} C_VEL
LIN {X 0,Y 298.645,Z 176.267,A -85,B 0,C 180,E1 -16374.599,E2 -16374.599} C_VEL
LIN {X 0,Y 298.912,Z 176.253,A -85,B 0,C 180,E1 -16378.653,E2 -16378.653} C_VEL
LIN {X 0,Y 298.912,Z 176.238,A -85,B 0,C 180,E1 -16381.347,E2 -16381.347} C_VEL
LIN {X 0,Y 298.786,Z 176.262,A -85,B 0,C 180,E1 -16386.754,E2 -16386.754} C_VEL
LIN {X 0,Y 298.671,Z 176.26,A -85,B 0,C 180,E1 -16389.481,E2 -16389.481} C_VEL
LIN {X 0,Y 298.542,Z 176.294,A -85,B 0,C 180,E1 -16393.616,E2 -16393.616} C_VEL
LIN {X 0,Y 298.539,Z 176.282,A -85,B 0,C 180,E1 -16396.409,E2 -16396.409} C_VEL
LIN {X 0,Y 298.503,Z 176.302,A -85,B 0,C 180,E1 -16399.655,E2 -16399.655} C_VEL
LIN {X 0,Y 298.449,Z 176.302,A -85,B 0,C 180,E1 -16403.599,E2 -16403.599} C_VEL
LIN {X 0,Y 298.479,Z 176.297,A -85,B 0,C 180,E1 -16406.576,E2 -16406.576} C_VEL
LIN {X 0,Y 298.413,Z 176.31,A -85,B 0,C 180,E1 -16409.642,E2 -16409.642} C_VEL
LIN {X 0,Y 298.388,Z 176.301,A -85,B 0,C 180,E1 -16412.801,E2 -16412.801} C_VEL
LIN {X 0,Y 298.44,Z 176.277,A -85,B 0,C 180,E1 -16416.809,E2 -16416.809} C_VEL
LIN {X 0,Y 298.382,Z 176.31,A -85,B 0,C 180,E1 -16421.089,E2 -16421.089} C_VEL
LIN {X 0,Y 298.394,Z 176.284,A -85,B 0,C 180,E1 -16423.105,E2 -16423.105} C_VEL
LIN {X 0,Y 298.398,Z 176.315,A -85,B 0,C 180,E1 -16426.922,E2 -16426.922} C_VEL
LIN {X 0,Y 298.395,Z 176.293,A -85,B 0,C 180,E1 -16431.009,E2 -16431.009} C_VEL
LIN {X 0,Y 298.415,Z 176.305,A -85,B 0,C 180,E1 -16433.931,E2 -16433.931} C_VEL
LIN {X 0,Y 298.393,Z 176.309,A -85,B 0,C 180,E1 -16437.985,E2 -16437.985} C_VEL
LIN {X 0,Y 298.443,Z 176.418,A -85,B 0,C 180,E1 -16438.798,E2 -16438.798} C_VEL
LIN {X 0,Y 300.538,Z 185.486,A -85,B 0,C 180,E1 -16442.117,E2 -16442.117} C_VEL
LIN {X 0,Y 301.14,Z 188.189,A -85,B 0,C 180,E1 -16442.961,E2 -16442.961} C_VEL
LIN {X 0,Y 308.111,Z 205.736,A -85,B 0,C 180,E1 -16444.11,E2 -16444.11} C_VEL
LIN {X 0,Y 311.52,Z 223.82,A -85,B 0,C 180,E1 -16444.868,E2 -16444.868} C_VEL
LIN {X 0,Y 309.768,Z 296.149,A -85,B 0,C 180,E1 -16446.564,E2 -16446.564} C_VEL
LIN {X 0,Y 308.808,Z 309.904,A -85,B 0,C 180,E1 -16447.151,E2 -16447.151} C_VEL
LIN {X 0,Y 307.763,Z 322.246,A -85,B 0,C 180,E1 -16447.954,E2 -16447.954} C_VEL
LIN {X 0,Y 306.375,Z 334.078,A -85,B 0,C 180,E1 -16448.998,E2 -16448.998} C_VEL
LIN {X 0,Y 304.802,Z 345.442,A -85,B 0,C 180,E1 -16450.294,E2 -16450.294} C_VEL
LIN {X 0,Y 303.4,Z 355.083,A -85,B 0,C 180,E1 -16451.678,E2 -16451.678} C_VEL
LIN {X 0,Y 301.907,Z 364.877,A -85,B 0,C 180,E1 -16453.432,E2 -16453.432} C_VEL
LIN {X 0,Y 300.25,Z 373.811,A -85,B 0,C 180,E1 -16455.427,E2 -16455.427} C_VEL
LIN {X 0,Y 299.025,Z 381.004,A -85,B 0,C 180,E1 -16457.444,E2 -16457.444} C_VEL
LIN {X 0,Y 298.168,Z 385.855,A -85,B 0,C 180,E1 -16459.132,E2 -16459.132} C_VEL
LIN {X 0,Y 297.424,Z 390.57,A -85,B 0,C 180,E1 -16461.166,E2 -16461.166} C_VEL
LIN {X 0,Y 296.947,Z 394.179,A -85,B 0,C 180,E1 -16463.205,E2 -16463.205} C_VEL
LIN {X 0,Y 296.748,Z 396.044,A -85,B 0,C 180,E1 -16464.565,E2 -16464.565} C_VEL
LIN {X 0,Y 296.64,Z 397.447,A -85,B 0,C 180,E1 -16465.925,E2 -16465.925} C_VEL
LIN {X 0,Y 296.555,Z 398.445,A -85,B 0,C 180,E1 -16467.284,E2 -16467.284} C_VEL
LIN {X 0,Y 296.454,Z 399.291,A -85,B 0,C 180,E1 -16470.001,E2 -16470.001} C_VEL
LIN {X 0,Y 296.463,Z 399.099,A -85,B 0,C 180,E1 -16471.359,E2 -16471.359} C_VEL
LIN {X 0,Y 296.554,Z 398.509,A -85,B 0,C 180,E1 -16472.717,E2 -16472.717} C_VEL
LIN {X 0,Y 296.634,Z 397.537,A -85,B 0,C 180,E1 -16474.076,E2 -16474.076} C_VEL
LIN {X 0,Y 296.83,Z 395.39,A -85,B 0,C 180,E1 -16476.048,E2 -16476.048} C_VEL
LIN {X 0,Y 297.269,Z 392.093,A -85,B 0,C 180,E1 -16478.155,E2 -16478.155} C_VEL
LIN {X 0,Y 297.855,Z 387.823,A -85,B 0,C 180,E1 -16480.193,E2 -16480.193} C_VEL
LIN {X 0,Y 298.983,Z 381.36,A -85,B 0,C 180,E1 -16482.559,E2 -16482.559} C_VEL
LIN {X 0,Y 300.199,Z 374.259,A -85,B 0,C 180,E1 -16484.577,E2 -16484.577} C_VEL
LIN {X 0,Y 301.809,Z 365.414,A -85,B 0,C 180,E1 -16486.574,E2 -16486.574} C_VEL
LIN {X 0,Y 303.178,Z 356.247,A -85,B 0,C 180,E1 -16488.254,E2 -16488.254} C_VEL
LIN {X 0,Y 304.703,Z 346.291,A -85,B 0,C 180,E1 -16489.714,E2 -16489.714} C_VEL
LIN {X 0,Y 306.321,Z 335.114,A -85,B 0,C 180,E1 -16491.007,E2 -16491.007} C_VEL
LIN {X 0,Y 307.742,Z 322.57,A -85,B 0,C 180,E1 -16492.137,E2 -16492.137} C_VEL
LIN {X 0,Y 308.911,Z 309.627,A -85,B 0,C 180,E1 -16492.974,E2 -16492.974} C_VEL
LIN {X 0,Y 309.783,Z 296.86,A -85,B 0,C 180,E1 -16493.525,E2 -16493.525} C_VEL
LIN {X 0,Y 310.631,Z 265.902,A -85,B 0,C 180,E1 -16494.277,E2 -16494.277} C_VEL
LIN {X 0,Y 311.48,Z 223.339,A -85,B 0,C 180,E1 -16495.265,E2 -16495.265} C_VEL
LIN {X 0,Y 308.148,Z 205.778,A -85,B 0,C 180,E1 -16496.004,E2 -16496.004} C_VEL
LIN {X 0,Y 301.137,Z 188.253,A -85,B 0,C 180,E1 -16497.155,E2 -16497.155} C_VEL
LIN {X 0,Y 300.359,Z 184.699,A -85,B 0,C 180,E1 -16498.283,E2 -16498.283} C_VEL
LIN {X 0,Y 298.503,Z 176.636,A -85,B 0,C 180,E1 -16501.196,E2 -16501.196} C_VEL
LIN {X 0,Y 298.415,Z 176.303,A -85,B 0,C 180,E1 -16501.782,E2 -16501.782} C_VEL
LIN {X 0,Y 298.432,Z 176.3,A -85,B 0,C 180,E1 -16506.068,E2 -16506.068} C_VEL
LIN {X 0,Y 298.403,Z 176.289,A -85,B 0,C 180,E1 -16509.487,E2 -16509.487} C_VEL
LIN {X 0,Y 298.398,Z 176.315,A -85,B 0,C 180,E1 -16513.103,E2 -16513.103} C_VEL
LIN {X 0,Y 298.402,Z 176.282,A -85,B 0,C 180,E1 -16516.92,E2 -16516.92} C_VEL
LIN {X 0,Y 298.378,Z 176.302,A -85,B 0,C 180,E1 -16518.654,E2 -16518.654} C_VEL
LIN {X 0,Y 297.766,Z 176.394,A -85,B 0,C 180,E1 -16519.781,E2 -16519.781} C_VEL
LIN {X 0,Y 294.928,Z 176.743,A -85,B 0,C 180,E1 -16521.615,E2 -16521.615} C_VEL
LIN {X 0,Y 292.488,Z 177.022,A -85,B 0,C 180,E1 -16523.104,E2 -16523.104} C_VEL
LIN {X 0,Y 291.442,Z 177.136,A -85,B 0,C 180,E1 -16524.258,E2 -16524.258} C_VEL
LIN {X 0,Y 291.359,Z 177.144,A -85,B 0,C 180,E1 -16524.649,E2 -16524.649} C_VEL
LIN {X 0,Y 291.37,Z 177.179,A -85,B 0,C 180,E1 -16527.95,E2 -16527.95} C_VEL
LIN {X 0,Y 291.38,Z 177.185,A -85,B 0,C 180,E1 -16531.158,E2 -16531.158} C_VEL
LIN {X 0,Y 291.411,Z 177.185,A -85,B 0,C 180,E1 -16534.271,E2 -16534.271} C_VEL
LIN {X 0,Y 291.371,Z 177.179,A -85,B 0,C 180,E1 -16537.299,E2 -16537.299} C_VEL
LIN {X 0,Y 291.455,Z 177.18,A -85,B 0,C 180,E1 -16540.27,E2 -16540.27} C_VEL
LIN {X 0,Y 291.538,Z 177.152,A -85,B 0,C 180,E1 -16544.634,E2 -16544.634} C_VEL
LIN {X 0,Y 291.533,Z 177.165,A -85,B 0,C 180,E1 -16548.88,E2 -16548.88} C_VEL
LIN {X 0,Y 291.706,Z 177.131,A -85,B 0,C 180,E1 -16551.688,E2 -16551.688} C_VEL
LIN {X 0,Y 291.623,Z 177.156,A -85,B 0,C 180,E1 -16554.468,E2 -16554.468} C_VEL
LIN {X 0,Y 291.884,Z 177.113,A -85,B 0,C 180,E1 -16558.62,E2 -16558.62} C_VEL
LIN {X 0,Y 291.883,Z 177.129,A -85,B 0,C 180,E1 -16561.38,E2 -16561.38} C_VEL
LIN {X 0,Y 291.718,Z 177.142,A -85,B 0,C 180,E1 -16566.919,E2 -16566.919} C_VEL
LIN {X 0,Y 291.564,Z 177.158,A -85,B 0,C 180,E1 -16569.714,E2 -16569.714} C_VEL
LIN {X 0,Y 291.511,Z 177.172,A -85,B 0,C 180,E1 -16573.951,E2 -16573.951} C_VEL
LIN {X 0,Y 291.437,Z 177.171,A -85,B 0,C 180,E1 -16576.821,E2 -16576.821} C_VEL
LIN {X 0,Y 291.421,Z 177.183,A -85,B 0,C 180,E1 -16579.86,E2 -16579.86} C_VEL
LIN {X 0,Y 291.379,Z 177.175,A -85,B 0,C 180,E1 -16584.207,E2 -16584.207} C_VEL
LIN {X 0,Y 291.417,Z 177.185,A -85,B 0,C 180,E1 -16587.272,E2 -16587.272} C_VEL
LIN {X 0,Y 291.331,Z 177.189,A -85,B 0,C 180,E1 -16590.438,E2 -16590.438} C_VEL
LIN {X 0,Y 291.342,Z 177.185,A -85,B 0,C 180,E1 -16593.699,E2 -16593.699} C_VEL
LIN {X 0,Y 291.373,Z 177.149,A -85,B 0,C 180,E1 -16597.254,E2 -16597.254} C_VEL
LIN {X 0,Y 291.331,Z 177.196,A -85,B 0,C 180,E1 -16600.643,E2 -16600.643} C_VEL
LIN {X 0,Y 291.289,Z 177.198,A -85,B 0,C 180,E1 -16604.402,E2 -16604.402} C_VEL
LIN {X 0,Y 291.325,Z 177.196,A -85,B 0,C 180,E1 -16608.405,E2 -16608.405} C_VEL
LIN {X 0,Y 291.338,Z 177.169,A -85,B 0,C 180,E1 -16611.156,E2 -16611.156} C_VEL
LIN {X 0,Y 291.361,Z 177.189,A -85,B 0,C 180,E1 -16614.626,E2 -16614.626} C_VEL
LIN {X 0,Y 291.412,Z 177.375,A -85,B 0,C 180,E1 -16616.73,E2 -16616.73} C_VEL
LIN {X 0,Y 293.814,Z 188.013,A -85,B 0,C 180,E1 -16620.636,E2 -16620.636} C_VEL
LIN {X 0,Y 294.803,Z 192.787,A -85,B 0,C 180,E1 -16622.23,E2 -16622.23} C_VEL
LIN {X 0,Y 297.835,Z 200.296,A -85,B 0,C 180,E1 -16622.793,E2 -16622.793} C_VEL
LIN {X 0,Y 300.716,Z 208.134,A -85,B 0,C 180,E1 -16623.28,E2 -16623.28} C_VEL
LIN {X 0,Y 305.019,Z 233.214,A -85,B 0,C 180,E1 -16624.329,E2 -16624.329} C_VEL
LIN {X 0,Y 303.213,Z 300.845,A -85,B 0,C 180,E1 -16625.934,E2 -16625.934} C_VEL
LIN {X 0,Y 302.243,Z 314.76,A -85,B 0,C 180,E1 -16626.534,E2 -16626.534} C_VEL
LIN {X 0,Y 300.975,Z 327.201,A -85,B 0,C 180,E1 -16627.338,E2 -16627.338} C_VEL
LIN {X 0,Y 299.663,Z 338.296,A -85,B 0,C 180,E1 -16628.322,E2 -16628.322} C_VEL
LIN {X 0,Y 298.007,Z 349.852,A -85,B 0,C 180,E1 -16629.644,E2 -16629.644} C_VEL
LIN {X 0,Y 296.315,Z 360.255,A -85,B 0,C 180,E1 -16631.146,E2 -16631.146} C_VEL
LIN {X 0,Y 294.815,Z 369.557,A -85,B 0,C 180,E1 -16632.829,E2 -16632.829} C_VEL
LIN {X 0,Y 293.324,Z 377.977,A -85,B 0,C 180,E1 -16634.718,E2 -16634.718} C_VEL
LIN {X 0,Y 291.898,Z 385.381,A -85,B 0,C 180,E1 -16636.777,E2 -16636.777} C_VEL
LIN {X 0,Y 290.874,Z 391.327,A -85,B 0,C 180,E1 -16638.855,E2 -16638.855} C_VEL
LIN {X 0,Y 290.149,Z 396.024,A -85,B 0,C 180,E1 -16640.941,E2 -16640.941} C_VEL
LIN {X 0,Y 289.71,Z 399.611,A -85,B 0,C 180,E1 -16643.033,E2 -16643.033} C_VEL
LIN {X 0,Y 289.517,Z 401.46,A -85,B 0,C 180,E1 -16644.427,E2 -16644.427} C_VEL
LIN {X 0,Y 289.423,Z 402.847,A -85,B 0,C 180,E1 -16645.822,E2 -16645.822} C_VEL
LIN {X 0,Y 289.399,Z 403.836,A -85,B 0,C 180,E1 -16647.216,E2 -16647.216} C_VEL
LIN {X 0,Y 289.373,Z 404.439,A -85,B 0,C 180,E1 -16648.608,E2 -16648.608} C_VEL
LIN {X 0,Y 289.372,Z 404.651,A -85,B 0,C 180,E1 -16649.999,E2 -16649.999} C_VEL
LIN {X 0,Y 289.373,Z 404.431,A -85,B 0,C 180,E1 -16651.391,E2 -16651.391} C_VEL
LIN {X 0,Y 289.399,Z 403.824,A -85,B 0,C 180,E1 -16652.783,E2 -16652.783} C_VEL
LIN {X 0,Y 289.556,Z 401.436,A -85,B 0,C 180,E1 -16655.571,E2 -16655.571} C_VEL
LIN {X 0,Y 289.847,Z 398.507,A -85,B 0,C 180,E1 -16657.663,E2 -16657.663} C_VEL
LIN {X 0,Y 290.357,Z 394.544,A -85,B 0,C 180,E1 -16659.754,E2 -16659.754} C_VEL
LIN {X 0,Y 291.362,Z 388.448,A -85,B 0,C 180,E1 -16662.184,E2 -16662.184} C_VEL
LIN {X 0,Y 292.577,Z 381.789,A -85,B 0,C 180,E1 -16664.253,E2 -16664.253} C_VEL
LIN {X 0,Y 294.086,Z 373.524,A -85,B 0,C 180,E1 -16666.307,E2 -16666.307} C_VEL
LIN {X 0,Y 295.505,Z 365.046,A -85,B 0,C 180,E1 -16668.009,E2 -16668.009} C_VEL
LIN {X 0,Y 297.2,Z 354.568,A -85,B 0,C 180,E1 -16669.692,E2 -16669.692} C_VEL
LIN {X 0,Y 298.771,Z 344.198,A -85,B 0,C 180,E1 -16671.021,E2 -16671.021} C_VEL
LIN {X 0,Y 300.33,Z 332.822,A -85,B 0,C 180,E1 -16672.168,E2 -16672.168} C_VEL
LIN {X 0,Y 301.628,Z 321.116,A -85,B 0,C 180,E1 -16673.061,E2 -16673.061} C_VEL
LIN {X 0,Y 302.654,Z 308.528,A -85,B 0,C 180,E1 -16673.749,E2 -16673.749} C_VEL
LIN {X 0,Y 303.385,Z 295.694,A -85,B 0,C 180,E1 -16674.187,E2 -16674.187} C_VEL
LIN {X 0,Y 304.895,Z 232.581,A -85,B 0,C 180,E1 -16675.669,E2 -16675.669} C_VEL
LIN {X 0,Y 300.497,Z 207.356,A -85,B 0,C 180,E1 -16676.73,E2 -16676.73} C_VEL
LIN {X 0,Y 294.842,Z 192.92,A -85,B 0,C 180,E1 -16677.715,E2 -16677.715} C_VEL
LIN {X 0,Y 293.75,Z 187.913,A -85,B 0,C 180,E1 -16679.37,E2 -16679.37} C_VEL
LIN {X 0,Y 291.391,Z 177.469,A -85,B 0,C 180,E1 -16683.183,E2 -16683.183} C_VEL
LIN {X 0,Y 291.354,Z 177.177,A -85,B 0,C 180,E1 -16683.696,E2 -16683.696} C_VEL
LIN {X 0,Y 291.363,Z 177.173,A -85,B 0,C 180,E1 -16687.25,E2 -16687.25} C_VEL
LIN {X 0,Y 291.326,Z 177.194,A -85,B 0,C 180,E1 -16690.642,E2 -16690.642} C_VEL
LIN {X 0,Y 291.285,Z 177.201,A -85,B 0,C 180,E1 -16694.401,E2 -16694.401} C_VEL
LIN {X 0,Y 291.32,Z 177.194,A -85,B 0,C 180,E1 -16698.403,E2 -16698.403} C_VEL
LIN {X 0,Y 291.346,Z 177.176,A -85,B 0,C 180,E1 -16701.157,E2 -16701.157} C_VEL
LIN {X 0,Y 291.354,Z 177.158,A -85,B 0,C 180,E1 -16704.625,E2 -16704.625} C_VEL
LIN {X 0,Y 291.363,Z 177.191,A -85,B 0,C 180,E1 -16707.95,E2 -16707.95} C_VEL
LIN {X 0,Y 291.369,Z 177.181,A -85,B 0,C 180,E1 -16711.157,E2 -16711.157} C_VEL
LIN {X 0,Y 291.405,Z 177.185,A -85,B 0,C 180,E1 -16714.271,E2 -16714.271} C_VEL
LIN {X 0,Y 291.365,Z 177.184,A -85,B 0,C 180,E1 -16717.298,E2 -16717.298} C_VEL
LIN {X 0,Y 291.45,Z 177.177,A -85,B 0,C 180,E1 -16720.27,E2 -16720.27} C_VEL
LIN {X 0,Y 291.488,Z 177.175,A -85,B 0,C 180,E1 -16724.665,E2 -16724.665} C_VEL
LIN {X 0,Y 291.528,Z 177.154,A -85,B 0,C 180,E1 -16728.88,E2 -16728.88} C_VEL
LIN {X 0,Y 291.696,Z 177.148,A -85,B 0,C 180,E1 -16731.688,E2 -16731.688} C_VEL
LIN {X 0,Y 291.616,Z 177.144,A -85,B 0,C 180,E1 -16734.468,E2 -16734.468} C_VEL
LIN {X 0,Y 291.879,Z 177.13,A -85,B 0,C 180,E1 -16738.62,E2 -16738.62} C_VEL
LIN {X 0,Y 291.879,Z 177.114,A -85,B 0,C 180,E1 -16741.38,E2 -16741.38} C_VEL
LIN {X 0,Y 291.735,Z 177.14,A -85,B 0,C 180,E1 -16746.918,E2 -16746.918} C_VEL
LIN {X 0,Y 291.62,Z 177.139,A -85,B 0,C 180,E1 -16749.712,E2 -16749.712} C_VEL
LIN {X 0,Y 291.512,Z 177.167,A -85,B 0,C 180,E1 -16753.951,E2 -16753.951} C_VEL
LIN {X 0,Y 291.478,Z 177.165,A -85,B 0,C 180,E1 -16756.819,E2 -16756.819} C_VEL
LIN {X 0,Y 291.443,Z 177.182,A -85,B 0,C 180,E1 -16759.876,E2 -16759.876} C_VEL
LIN {X 0,Y 291.392,Z 177.186,A -85,B 0,C 180,E1 -16764.206,E2 -16764.206} C_VEL
LIN {X 0,Y 291.414,Z 177.174,A -85,B 0,C 180,E1 -16767.273,E2 -16767.273} C_VEL
LIN {X 0,Y 291.33,Z 177.197,A -85,B 0,C 180,E1 -16770.438,E2 -16770.438} C_VEL
LIN {X 0,Y 291.337,Z 177.159,A -85,B 0,C 180,E1 -16773.7,E2 -16773.7} C_VEL
LIN {X 0,Y 291.369,Z 177.166,A -85,B 0,C 180,E1 -16777.255,E2 -16777.255} C_VEL
LIN {X 0,Y 291.327,Z 177.192,A -85,B 0,C 180,E1 -16780.644,E2 -16780.644} C_VEL
LIN {X 0,Y 291.285,Z 177.173,A -85,B 0,C 180,E1 -16784.403,E2 -16784.403} C_VEL
LIN {X 0,Y 291.322,Z 177.184,A -85,B 0,C 180,E1 -16788.406,E2 -16788.406} C_VEL
LIN {X 0,Y 291.344,Z 177.172,A -85,B 0,C 180,E1 -16791.159,E2 -16791.159} C_VEL
LIN {X 0,Y 291.358,Z 177.176,A -85,B 0,C 180,E1 -16794.627,E2 -16794.627} C_VEL
LIN {X 0,Y 291.411,Z 177.321,A -85,B 0,C 180,E1 -16798.262,E2 -16798.262} C_VEL
LIN {X 0,Y 293.682,Z 187.143,A -85,B 0,C 180,E1 -16801.937,E2 -16801.937} C_VEL
LIN {X 0,Y 293.984,Z 188.515,A -85,B 0,C 180,E1 -16802.274,E2 -16802.274} C_VEL
LIN {X 0,Y 301.482,Z 206.833,A -85,B 0,C 180,E1 -16803.524,E2 -16803.524} C_VEL
LIN {X 0,Y 302.604,Z 211.067,A -85,B 0,C 180,E1 -16803.74,E2 -16803.74} C_VEL
LIN {X 0,Y 305.084,Z 225.82,A -85,B 0,C 180,E1 -16804.348,E2 -16804.348} C_VEL
LIN {X 0,Y 303.273,Z 296.23,A -85,B 0,C 180,E1 -16806.031,E2 -16806.031} C_VEL
LIN {X 0,Y 302.297,Z 309.979,A -85,B 0,C 180,E1 -16806.63,E2 -16806.63} C_VEL
LIN {X 0,Y 301.216,Z 322.317,A -85,B 0,C 180,E1 -16807.449,E2 -16807.449} C_VEL
LIN {X 0,Y 299.767,Z 334.148,A -85,B 0,C 180,E1 -16808.512,E2 -16808.512} C_VEL
LIN {X 0,Y 298.113,Z 345.512,A -85,B 0,C 180,E1 -16809.833,E2 -16809.833} C_VEL
LIN {X 0,Y 296.593,Z 355.522,A -85,B 0,C 180,E1 -16811.305,E2 -16811.305} C_VEL
LIN {X 0,Y 295.086,Z 364.945,A -85,B 0,C 180,E1 -16813.038,E2 -16813.038} C_VEL
LIN {X 0,Y 293.384,Z 373.879,A -85,B 0,C 180,E1 -16815.078,E2 -16815.078} C_VEL
LIN {X 0,Y 292.06,Z 381.071,A -85,B 0,C 180,E1 -16817.14,E2 -16817.14} C_VEL
LIN {X 0,Y 291.193,Z 385.922,A -85,B 0,C 180,E1 -16818.868,E2 -16818.868} C_VEL
LIN {X 0,Y 290.399,Z 390.637,A -85,B 0,C 180,E1 -16820.95,E2 -16820.95} C_VEL
LIN {X 0,Y 289.887,Z 394.245,A -85,B 0,C 180,E1 -16823.038,E2 -16823.038} C_VEL
LIN {X 0,Y 289.674,Z 396.11,A -85,B 0,C 180,E1 -16824.432,E2 -16824.432} C_VEL
LIN {X 0,Y 289.545,Z 397.512,A -85,B 0,C 180,E1 -16825.825,E2 -16825.825} C_VEL
LIN {X 0,Y 289.464,Z 398.51,A -85,B 0,C 180,E1 -16827.217,E2 -16827.217} C_VEL
LIN {X 0,Y 289.374,Z 399.356,A -85,B 0,C 180,E1 -16830.001,E2 -16830.001} C_VEL
LIN {X 0,Y 289.387,Z 399.163,A -85,B 0,C 180,E1 -16831.392,E2 -16831.392} C_VEL
LIN {X 0,Y 289.462,Z 398.574,A -85,B 0,C 180,E1 -16832.784,E2 -16832.784} C_VEL
LIN {X 0,Y 289.538,Z 397.602,A -85,B 0,C 180,E1 -16834.176,E2 -16834.176} C_VEL
LIN {X 0,Y 289.749,Z 395.674,A -85,B 0,C 180,E1 -16836.024,E2 -16836.024} C_VEL
LIN {X 0,Y 290.21,Z 392.157,A -85,B 0,C 180,E1 -16838.355,E2 -16838.355} C_VEL
LIN {X 0,Y 290.865,Z 387.887,A -85,B 0,C 180,E1 -16840.441,E2 -16840.441} C_VEL
LIN {X 0,Y 292.013,Z 381.423,A -85,B 0,C 180,E1 -16842.863,E2 -16842.863} C_VEL
LIN {X 0,Y 293.332,Z 374.322,A -85,B 0,C 180,E1 -16844.926,E2 -16844.926} C_VEL
LIN {X 0,Y 294.988,Z 365.476,A -85,B 0,C 180,E1 -16846.969,E2 -16846.969} C_VEL
LIN {X 0,Y 296.414,Z 356.406,A -85,B 0,C 180,E1 -16848.668,E2 -16848.668} C_VEL
LIN {X 0,Y 298.02,Z 346.352,A -85,B 0,C 180,E1 -16850.175,E2 -16850.175} C_VEL
LIN {X 0,Y 299.709,Z 335.173,A -85,B 0,C 180,E1 -16851.494,E2 -16851.494} C_VEL
LIN {X 0,Y 301.186,Z 322.628,A -85,B 0,C 180,E1 -16852.645,E2 -16852.645} C_VEL
LIN {X 0,Y 302.393,Z 309.682,A -85,B 0,C 180,E1 -16853.499,E2 -16853.499} C_VEL
LIN {X 0,Y 303.294,Z 296.91,A -85,B 0,C 180,E1 -16854.06,E2 -16854.06} C_VEL
LIN {X 0,Y 304.174,Z 265.816,A -85,B 0,C 180,E1 -16854.83,E2 -16854.83} C_VEL
LIN {X 0,Y 305.123,Z 224.719,A -85,B 0,C 180,E1 -16855.796,E2 -16855.796} C_VEL
LIN {X 0,Y 301.927,Z 208.097,A -85,B 0,C 180,E1 -16856.522,E2 -16856.522} C_VEL
LIN {X 0,Y 295.282,Z 191.546,A -85,B 0,C 180,E1 -16857.613,E2 -16857.613} C_VEL
LIN {X 0,Y 293.887,Z 188.133,A -85,B 0,C 180,E1 -16857.905,E2 -16857.905} C_VEL
LIN {X 0,Y 291.81,Z 178.987,A -85,B 0,C 180,E1 -16861.185,E2 -16861.185} C_VEL
LIN {X 0,Y 291.362,Z 177.208,A -85,B 0,C 180,E1 -16861.999,E2 -16861.999} C_VEL
LIN {X 0,Y 291.386,Z 177.171,A -85,B 0,C 180,E1 -16865.37,E2 -16865.37} C_VEL
LIN {X 0,Y 291.354,Z 177.173,A -85,B 0,C 180,E1 -16868.841,E2 -16868.841} C_VEL
LIN {X 0,Y 291.32,Z 177.193,A -85,B 0,C 180,E1 -16872.492,E2 -16872.492} C_VEL
LIN {X 0,Y 291.308,Z 177.165,A -85,B 0,C 180,E1 -16876.366,E2 -16876.366} C_VEL
LIN {X 0,Y 291.38,Z 177.19,A -85,B 0,C 180,E1 -16880.518,E2 -16880.518} C_VEL
LIN {X 0,Y 291.406,Z 177.161,A -85,B 0,C 180,E1 -16882.919,E2 -16882.919} C_VEL
LIN {X 0,Y 291.359,Z 177.144,A -85,B 0,C 180,E1 -16884.649,E2 -16884.649} C_VEL
LIN {X 0,Y 290.709,Z 177.23,A -85,B 0,C 180,E1 -16885.802,E2 -16885.802} C_VEL
LIN {X 0,Y 287.895,Z 177.609,A -85,B 0,C 180,E1 -16887.682,E2 -16887.682} C_VEL
LIN {X 0,Y 285.486,Z 177.922,A -85,B 0,C 180,E1 -16889.207,E2 -16889.207} C_VEL
LIN {X 0,Y 284.427,Z 178.053,A -85,B 0,C 180,E1 -16890.389,E2 -16890.389} C_VEL
LIN {X 0,Y 284.328,Z 178.06,A -85,B 0,C 180,E1 -16890.789,E2 -16890.789} C_VEL
LIN {X 0,Y 284.374,Z 178.054,A -85,B 0,C 180,E1 -16893.586,E2 -16893.586} C_VEL
LIN {X 0,Y 284.33,Z 178.061,A -85,B 0,C 180,E1 -16896.704,E2 -16896.704} C_VEL
LIN {X 0,Y 284.396,Z 178.059,A -85,B 0,C 180,E1 -16901.261,E2 -16901.261} C_VEL
LIN {X 0,Y 284.475,Z 178.031,A -85,B 0,C 180,E1 -16904.47,E2 -16904.47} C_VEL
LIN {X 0,Y 284.485,Z 178.043,A -85,B 0,C 180,E1 -16908.601,E2 -16908.601} C_VEL
LIN {X 0,Y 284.656,Z 178.007,A -85,B 0,C 180,E1 -16911.481,E2 -16911.481} C_VEL
LIN {X 0,Y 284.594,Z 178.032,A -85,B 0,C 180,E1 -16914.331,E2 -16914.331} C_VEL
LIN {X 0,Y 284.85,Z 177.988,A -85,B 0,C 180,E1 -16918.586,E2 -16918.586} C_VEL
LIN {X 0,Y 284.849,Z 178.005,A -85,B 0,C 180,E1 -16921.414,E2 -16921.414} C_VEL
LIN {X 0,Y 284.669,Z 178.022,A -85,B 0,C 180,E1 -16927.091,E2 -16927.091} C_VEL
LIN {X 0,Y 284.51,Z 178.035,A -85,B 0,C 180,E1 -16929.957,E2 -16929.957} C_VEL
LIN {X 0,Y 284.459,Z 178.05,A -85,B 0,C 180,E1 -16934.304,E2 -16934.304} C_VEL
LIN {X 0,Y 284.378,Z 178.048,A -85,B 0,C 180,E1 -16938.74,E2 -16938.74} C_VEL
LIN {X 0,Y 284.313,Z 178.067,A -85,B 0,C 180,E1 -16941.764,E2 -16941.764} C_VEL
LIN {X 0,Y 284.335,Z 178.056,A -85,B 0,C 180,E1 -16944.847,E2 -16944.847} C_VEL
LIN {X 0,Y 284.325,Z 178.064,A -85,B 0,C 180,E1 -16948.011,E2 -16948.011} C_VEL
LIN {X 0,Y 284.291,Z 178.072,A -85,B 0,C 180,E1 -16951.275,E2 -16951.275} C_VEL
LIN {X 0,Y 284.339,Z 178.03,A -85,B 0,C 180,E1 -16955.348,E2 -16955.348} C_VEL
LIN {X 0,Y 284.31,Z 178.039,A -85,B 0,C 180,E1 -16958.169,E2 -16958.169} C_VEL
LIN {X 0,Y 284.268,Z 178.069,A -85,B 0,C 180,E1 -16962.125,E2 -16962.125} C_VEL
LIN {X 0,Y 284.254,Z 178.073,A -85,B 0,C 180,E1 -16966.19,E2 -16966.19} C_VEL
LIN {X 0,Y 284.306,Z 178.057,A -85,B 0,C 180,E1 -16970.024,E2 -16970.024} C_VEL
LIN {X 0,Y 284.328,Z 178.064,A -85,B 0,C 180,E1 -16973.614,E2 -16973.614} C_VEL
LIN {X 0,Y 284.374,Z 178.204,A -85,B 0,C 180,E1 -16976.11,E2 -16976.11} C_VEL
LIN {X 0,Y 286.579,Z 188.111,A -85,B 0,C 180,E1 -16979.877,E2 -16979.877} C_VEL
LIN {X 0,Y 287.579,Z 192.751,A -85,B 0,C 180,E1 -16981.474,E2 -16981.474} C_VEL
LIN {X 0,Y 291.308,Z 201.791,A -85,B 0,C 180,E1 -16982.173,E2 -16982.173} C_VEL
LIN {X 0,Y 294.458,Z 209.845,A -85,B 0,C 180,E1 -16982.712,E2 -16982.712} C_VEL
LIN {X 0,Y 298.603,Z 233.927,A -85,B 0,C 180,E1 -16983.755,E2 -16983.755} C_VEL
LIN {X 0,Y 296.759,Z 300.794,A -85,B 0,C 180,E1 -16985.376,E2 -16985.376} C_VEL
LIN {X 0,Y 295.756,Z 314.704,A -85,B 0,C 180,E1 -16985.987,E2 -16985.987} C_VEL
LIN {X 0,Y 294.432,Z 327.143,A -85,B 0,C 180,E1 -16986.806,E2 -16986.806} C_VEL
LIN {X 0,Y 293.074,Z 338.235,A -85,B 0,C 180,E1 -16987.809,E2 -16987.809} C_VEL
LIN {X 0,Y 291.371,Z 349.791,A -85,B 0,C 180,E1 -16989.159,E2 -16989.159} C_VEL
LIN {X 0,Y 289.579,Z 360.193,A -85,B 0,C 180,E1 -16990.69,E2 -16990.69} C_VEL
LIN {X 0,Y 287.962,Z 369.821,A -85,B 0,C 180,E1 -16992.481,E2 -16992.481} C_VEL
LIN {X 0,Y 286.452,Z 377.914,A -85,B 0,C 180,E1 -16994.343,E2 -16994.343} C_VEL
LIN {X 0,Y 284.945,Z 385.318,A -85,B 0,C 180,E1 -16996.449,E2 -16996.449} C_VEL
LIN {X 0,Y 283.9,Z 391.263,A -85,B 0,C 180,E1 -16998.577,E2 -16998.577} C_VEL
LIN {X 0,Y 283.118,Z 395.96,A -85,B 0,C 180,E1 -17000.714,E2 -17000.714} C_VEL
LIN {X 0,Y 282.658,Z 399.547,A -85,B 0,C 180,E1 -17002.858,E2 -17002.858} C_VEL
LIN {X 0,Y 282.426,Z 401.605,A -85,B 0,C 180,E1 -17004.489,E2 -17004.489} C_VEL
LIN {X 0,Y 282.31,Z 403.772,A -85,B 0,C 180,E1 -17007.146,E2 -17007.146} C_VEL
LIN {X 0,Y 282.298,Z 404.375,A -85,B 0,C 180,E1 -17008.573,E2 -17008.573} C_VEL
LIN {X 0,Y 282.294,Z 404.586,A -85,B 0,C 180,E1 -17009.999,E2 -17009.999} C_VEL
LIN {X 0,Y 282.298,Z 404.366,A -85,B 0,C 180,E1 -17011.426,E2 -17011.426} C_VEL
LIN {X 0,Y 282.31,Z 403.759,A -85,B 0,C 180,E1 -17012.853,E2 -17012.853} C_VEL
LIN {X 0,Y 282.483,Z 401.37,A -85,B 0,C 180,E1 -17015.711,E2 -17015.711} C_VEL
LIN {X 0,Y 282.782,Z 398.441,A -85,B 0,C 180,E1 -17017.856,E2 -17017.856} C_VEL
LIN {X 0,Y 283.346,Z 394.478,A -85,B 0,C 180,E1 -17019.998,E2 -17019.998} C_VEL
LIN {X 0,Y 284.389,Z 388.381,A -85,B 0,C 180,E1 -17022.487,E2 -17022.487} C_VEL
LIN {X 0,Y 285.692,Z 381.722,A -85,B 0,C 180,E1 -17024.604,E2 -17024.604} C_VEL
LIN {X 0,Y 287.233,Z 373.457,A -85,B 0,C 180,E1 -17026.707,E2 -17026.707} C_VEL
LIN {X 0,Y 288.748,Z 364.978,A -85,B 0,C 180,E1 -17028.445,E2 -17028.445} C_VEL
LIN {X 0,Y 290.518,Z 354.5,A -85,B 0,C 180,E1 -17030.164,E2 -17030.164} C_VEL
LIN {X 0,Y 292.16,Z 344.129,A -85,B 0,C 180,E1 -17031.52,E2 -17031.52} C_VEL
LIN {X 0,Y 293.769,Z 332.752,A -85,B 0,C 180,E1 -17032.69,E2 -17032.69} C_VEL
LIN {X 0,Y 295.112,Z 321.043,A -85,B 0,C 180,E1 -17033.601,E2 -17033.601} C_VEL
LIN {X 0,Y 296.268,Z 307.538,A -85,B 0,C 180,E1 -17034.34,E2 -17034.34} C_VEL
LIN {X 0,Y 296.975,Z 294.023,A -85,B 0,C 180,E1 -17034.79,E2 -17034.79} C_VEL
LIN {X 0,Y 298.487,Z 233.711,A -85,B 0,C 180,E1 -17036.23,E2 -17036.23} C_VEL
LIN {X 0,Y 294.376,Z 209.62,A -85,B 0,C 180,E1 -17037.269,E2 -17037.269} C_VEL
LIN {X 0,Y 287.634,Z 192.935,A -85,B 0,C 180,E1 -17038.459,E2 -17038.459} C_VEL
LIN {X 0,Y 286.797,Z 189.116,A -85,B 0,C 180,E1 -17039.721,E2 -17039.721} C_VEL
LIN {X 0,Y 284.622,Z 179.465,A -85,B 0,C 180,E1 -17043.324,E2 -17043.324} C_VEL
LIN {X 0,Y 284.302,Z 178.076,A -85,B 0,C 180,E1 -17044.005,E2 -17044.005} C_VEL
LIN {X 0,Y 284.31,Z 178.046,A -85,B 0,C 180,E1 -17047.719,E2 -17047.719} C_VEL
LIN {X 0,Y 284.301,Z 178.059,A -85,B 0,C 180,E1 -17049.994,E2 -17049.994} C_VEL
LIN {X 0,Y 284.241,Z 178.078,A -85,B 0,C 180,E1 -17054.189,E2 -17054.189} C_VEL
LIN {X 0,Y 284.266,Z 178.072,A -85,B 0,C 180,E1 -17058.123,E2 -17058.123} C_VEL
LIN {X 0,Y 284.315,Z 178.031,A -85,B 0,C 180,E1 -17062.277,E2 -17062.277} C_VEL
LIN {X 0,Y 284.301,Z 178.046,A -85,B 0,C 180,E1 -17065.35,E2 -17065.35} C_VEL
LIN {X 0,Y 284.286,Z 178.072,A -85,B 0,C 180,E1 -17068.724,E2 -17068.724} C_VEL
LIN {X 0,Y 284.387,Z 178.061,A -85,B 0,C 180,E1 -17072.826,E2 -17072.826} C_VEL
LIN {X 0,Y 284.324,Z 178.055,A -85,B 0,C 180,E1 -17076.703,E2 -17076.703} C_VEL
LIN {X 0,Y 284.368,Z 178.061,A -85,B 0,C 180,E1 -17079.904,E2 -17079.904} C_VEL
LIN {X 0,Y 284.438,Z 178.052,A -85,B 0,C 180,E1 -17084.492,E2 -17084.492} C_VEL
LIN {X 0,Y 284.479,Z 178.031,A -85,B 0,C 180,E1 -17088.601,E2 -17088.601} C_VEL
LIN {X 0,Y 284.647,Z 178.027,A -85,B 0,C 180,E1 -17091.481,E2 -17091.481} C_VEL
LIN {X 0,Y 284.587,Z 178.02,A -85,B 0,C 180,E1 -17094.331,E2 -17094.331} C_VEL
LIN {X 0,Y 284.845,Z 178.005,A -85,B 0,C 180,E1 -17098.586,E2 -17098.586} C_VEL
LIN {X 0,Y 284.845,Z 177.989,A -85,B 0,C 180,E1 -17101.414,E2 -17101.414} C_VEL
LIN {X 0,Y 284.688,Z 178.017,A -85,B 0,C 180,E1 -17107.09,E2 -17107.09} C_VEL
LIN {X 0,Y 284.557,Z 178.02,A -85,B 0,C 180,E1 -17109.956,E2 -17109.956} C_VEL
LIN {X 0,Y 284.469,Z 178.04,A -85,B 0,C 180,E1 -17114.304,E2 -17114.304} C_VEL
LIN {X 0,Y 284.416,Z 178.05,A -85,B 0,C 180,E1 -17117.249,E2 -17117.249} C_VEL
LIN {X 0,Y 284.371,Z 178.058,A -85,B 0,C 180,E1 -17120.243,E2 -17120.243} C_VEL
LIN {X 0,Y 284.361,Z 178.059,A -85,B 0,C 180,E1 -17123.876,E2 -17123.876} C_VEL
LIN {X 0,Y 284.389,Z 178.049,A -85,B 0,C 180,E1 -17127.174,E2 -17127.174} C_VEL
LIN {X 0,Y 284.289,Z 178.071,A -85,B 0,C 180,E1 -17131.275,E2 -17131.275} C_VEL
LIN {X 0,Y 284.334,Z 178.018,A -85,B 0,C 180,E1 -17135.349,E2 -17135.349} C_VEL
LIN {X 0,Y 284.306,Z 178.06,A -85,B 0,C 180,E1 -17138.17,E2 -17138.17} C_VEL
LIN {X 0,Y 284.264,Z 178.051,A -85,B 0,C 180,E1 -17142.126,E2 -17142.126} C_VEL
LIN {X 0,Y 284.251,Z 178.074,A -85,B 0,C 180,E1 -17146.191,E2 -17146.191} C_VEL
LIN {X 0,Y 284.303,Z 178.042,A -85,B 0,C 180,E1 -17150.025,E2 -17150.025} C_VEL
LIN {X 0,Y 284.327,Z 178.063,A -85,B 0,C 180,E1 -17153.615,E2 -17153.615} C_VEL
LIN {X 0,Y 284.351,Z 178.293,A -85,B 0,C 180,E1 -17157.726,E2 -17157.726} C_VEL
LIN {X 0,Y 286.575,Z 187.736,A -85,B 0,C 180,E1 -17161.33,E2 -17161.33} C_VEL
LIN {X 0,Y 286.898,Z 188.866,A -85,B 0,C 180,E1 -17161.539,E2 -17161.539} C_VEL
LIN {X 0,Y 294.425,Z 206.769,A -85,B 0,C 180,E1 -17162.833,E2 -17162.833} C_VEL
LIN {X 0,Y 296.26,Z 212.194,A -85,B 0,C 180,E1 -17163.16,E2 -17163.16} C_VEL
LIN {X 0,Y 298.66,Z 225.781,A -85,B 0,C 180,E1 -17163.752,E2 -17163.752} C_VEL
LIN {X 0,Y 296.816,Z 296.31,A -85,B 0,C 180,E1 -17165.475,E2 -17165.475} C_VEL
LIN {X 0,Y 295.805,Z 310.054,A -85,B 0,C 180,E1 -17166.086,E2 -17166.086} C_VEL
LIN {X 0,Y 294.686,Z 322.389,A -85,B 0,C 180,E1 -17166.921,E2 -17166.921} C_VEL
LIN {X 0,Y 293.182,Z 334.218,A -85,B 0,C 180,E1 -17168.004,E2 -17168.004} C_VEL
LIN {X 0,Y 291.45,Z 345.581,A -85,B 0,C 180,E1 -17169.351,E2 -17169.351} C_VEL
LIN {X 0,Y 289.765,Z 356.222,A -85,B 0,C 180,E1 -17170.962,E2 -17170.962} C_VEL
LIN {X 0,Y 288.28,Z 365.013,A -85,B 0,C 180,E1 -17172.625,E2 -17172.625} C_VEL
LIN {X 0,Y 286.532,Z 373.946,A -85,B 0,C 180,E1 -17174.713,E2 -17174.713} C_VEL
LIN {X 0,Y 285.123,Z 381.138,A -85,B 0,C 180,E1 -17176.821,E2 -17176.821} C_VEL
LIN {X 0,Y 284.228,Z 385.988,A -85,B 0,C 180,E1 -17178.592,E2 -17178.592} C_VEL
LIN {X 0,Y 283.389,Z 390.703,A -85,B 0,C 180,E1 -17180.724,E2 -17180.724} C_VEL
LIN {X 0,Y 282.819,Z 394.311,A -85,B 0,C 180,E1 -17182.863,E2 -17182.863} C_VEL
LIN {X 0,Y 282.611,Z 396.175,A -85,B 0,C 180,E1 -17184.292,E2 -17184.292} C_VEL
LIN {X 0,Y 282.453,Z 397.578,A -85,B 0,C 180,E1 -17185.72,E2 -17185.72} C_VEL
LIN {X 0,Y 282.375,Z 398.575,A -85,B 0,C 180,E1 -17187.147,E2 -17187.147} C_VEL
LIN {X 0,Y 282.313,Z 399.189,A -85,B 0,C 180,E1 -17188.574,E2 -17188.574} C_VEL
LIN {X 0,Y 282.297,Z 399.421,A -85,B 0,C 180,E1 -17190.001,E2 -17190.001} C_VEL
LIN {X 0,Y 282.313,Z 399.228,A -85,B 0,C 180,E1 -17191.427,E2 -17191.427} C_VEL
LIN {X 0,Y 282.374,Z 398.639,A -85,B 0,C 180,E1 -17192.854,E2 -17192.854} C_VEL
LIN {X 0,Y 282.592,Z 396.302,A -85,B 0,C 180,E1 -17195.71,E2 -17195.71} C_VEL
LIN {X 0,Y 283.001,Z 393.421,A -85,B 0,C 180,E1 -17197.851,E2 -17197.851} C_VEL
LIN {X 0,Y 283.613,Z 389.515,A -85,B 0,C 180,E1 -17199.99,E2 -17199.99} C_VEL
LIN {X 0,Y 284.509,Z 384.478,A -85,B 0,C 180,E1 -17202.121,E2 -17202.121} C_VEL
LIN {X 0,Y 285.675,Z 378.136,A -85,B 0,C 180,E1 -17204.242,E2 -17204.242} C_VEL
LIN {X 0,Y 287.293,Z 370.201,A -85,B 0,C 180,E1 -17206.339,E2 -17206.339} C_VEL
LIN {X 0,Y 288.75,Z 362.207,A -85,B 0,C 180,E1 -17208.06,E2 -17208.06} C_VEL
LIN {X 0,Y 290.355,Z 352.249,A -85,B 0,C 180,E1 -17209.808,E2 -17209.808} C_VEL
LIN {X 0,Y 292.222,Z 341.147,A -85,B 0,C 180,E1 -17211.331,E2 -17211.331} C_VEL
LIN {X 0,Y 293.786,Z 330.264,A -85,B 0,C 180,E1 -17212.504,E2 -17212.504} C_VEL
LIN {X 0,Y 295.142,Z 318.24,A -85,B 0,C 180,E1 -17213.507,E2 -17213.507} C_VEL
LIN {X 0,Y 296.208,Z 305.888,A -85,B 0,C 180,E1 -17214.253,E2 -17214.253} C_VEL
LIN {X 0,Y 296.994,Z 293.086,A -85,B 0,C 180,E1 -17214.743,E2 -17214.743} C_VEL
LIN {X 0,Y 298.663,Z 225.292,A -85,B 0,C 180,E1 -17216.382,E2 -17216.382} C_VEL
LIN {X 0,Y 295.714,Z 210.139,A -85,B 0,C 180,E1 -17217.071,E2 -17217.071} C_VEL
LIN {X 0,Y 287.922,Z 191.163,A -85,B 0,C 180,E1 -17218.394,E2 -17218.394} C_VEL
LIN {X 0,Y 286.648,Z 188.096,A -85,B 0,C 180,E1 -17218.692,E2 -17218.692} C_VEL
LIN {X 0,Y 284.831,Z 180.212,A -85,B 0,C 180,E1 -17221.623,E2 -17221.623} C_VEL
LIN {X 0,Y 284.319,Z 178.087,A -85,B 0,C 180,E1 -17222.565,E2 -17222.565} C_VEL
LIN {X 0,Y 284.348,Z 178.057,A -85,B 0,C 180,E1 -17226.383,E2 -17226.383} C_VEL
LIN {X 0,Y 284.306,Z 178.041,A -85,B 0,C 180,E1 -17229.994,E2 -17229.994} C_VEL
LIN {X 0,Y 284.246,Z 178.073,A -85,B 0,C 180,E1 -17234.19,E2 -17234.19} C_VEL
LIN {X 0,Y 284.271,Z 178.05,A -85,B 0,C 180,E1 -17238.124,E2 -17238.124} C_VEL
LIN {X 0,Y 284.321,Z 178.056,A -85,B 0,C 180,E1 -17242.278,E2 -17242.278} C_VEL
LIN {X 0,Y 284.307,Z 178.021,A -85,B 0,C 180,E1 -17245.35,E2 -17245.35} C_VEL
LIN {X 0,Y 284.294,Z 178.071,A -85,B 0,C 180,E1 -17248.725,E2 -17248.725} C_VEL
LIN {X 0,Y 284.328,Z 178.06,A -85,B 0,C 180,E1 -17250.789,E2 -17250.789} C_VEL
LIN {X 0,Y 283.624,Z 178.144,A -85,B 0,C 180,E1 -17251.972,E2 -17251.972} C_VEL
LIN {X 0,Y 280.76,Z 178.507,A -85,B 0,C 180,E1 -17253.898,E2 -17253.898} C_VEL
LIN {X 0,Y 278.356,Z 178.813,A -85,B 0,C 180,E1 -17255.462,E2 -17255.462} C_VEL
LIN {X 0,Y 277.332,Z 178.933,A -85,B 0,C 180,E1 -17256.674,E2 -17256.674} C_VEL
LIN {X 0,Y 277.252,Z 178.936,A -85,B 0,C 180,E1 -17257.085,E2 -17257.085} C_VEL
LIN {X 0,Y 277.34,Z 178.937,A -85,B 0,C 180,E1 -17260.766,E2 -17260.766} C_VEL
LIN {X 0,Y 277.425,Z 178.913,A -85,B 0,C 180,E1 -17265.325,E2 -17265.325} C_VEL
LIN {X 0,Y 277.504,Z 178.901,A -85,B 0,C 180,E1 -17269.788,E2 -17269.788} C_VEL
LIN {X 0,Y 277.649,Z 178.893,A -85,B 0,C 180,E1 -17272.729,E2 -17272.729} C_VEL
LIN {X 0,Y 277.816,Z 178.863,A -85,B 0,C 180,E1 -17278.55,E2 -17278.55} C_VEL
LIN {X 0,Y 277.815,Z 178.881,A -85,B 0,C 180,E1 -17281.45,E2 -17281.45} C_VEL
LIN {X 0,Y 277.623,Z 178.9,A -85,B 0,C 180,E1 -17287.272,E2 -17287.272} C_VEL
LIN {X 0,Y 277.451,Z 178.913,A -85,B 0,C 180,E1 -17290.213,E2 -17290.213} C_VEL
LIN {X 0,Y 277.406,Z 178.929,A -85,B 0,C 180,E1 -17294.676,E2 -17294.676} C_VEL
LIN {X 0,Y 277.325,Z 178.93,A -85,B 0,C 180,E1 -17299.235,E2 -17299.235} C_VEL
LIN {X 0,Y 277.294,Z 178.928,A -85,B 0,C 180,E1 -17303.924,E2 -17303.924} C_VEL
LIN {X 0,Y 277.321,Z 178.938,A -85,B 0,C 180,E1 -17307.504,E2 -17307.504} C_VEL
LIN {X 0,Y 277.27,Z 178.94,A -85,B 0,C 180,E1 -17310.482,E2 -17310.482} C_VEL
LIN {X 0,Y 277.245,Z 178.937,A -85,B 0,C 180,E1 -17313.896,E2 -17313.896} C_VEL
LIN {X 0,Y 277.265,Z 178.906,A -85,B 0,C 180,E1 -17317.47,E2 -17317.47} C_VEL
LIN {X 0,Y 277.208,Z 178.954,A -85,B 0,C 180,E1 -17321.237,E2 -17321.237} C_VEL
LIN {X 0,Y 277.2,Z 178.957,A -85,B 0,C 180,E1 -17325.227,E2 -17325.227} C_VEL
LIN {X 0,Y 277.222,Z 178.948,A -85,B 0,C 180,E1 -17329.512,E2 -17329.512} C_VEL
LIN {X 0,Y 277.26,Z 178.926,A -85,B 0,C 180,E1 -17332.53,E2 -17332.53} C_VEL
LIN {X 0,Y 277.293,Z 179.056,A -85,B 0,C 180,E1 -17335.452,E2 -17335.452} C_VEL
LIN {X 0,Y 279.273,Z 187.541,A -85,B 0,C 180,E1 -17338.829,E2 -17338.829} C_VEL
LIN {X 0,Y 280.359,Z 192.659,A -85,B 0,C 180,E1 -17340.666,E2 -17340.666} C_VEL
LIN {X 0,Y 283.499,Z 199.975,A -85,B 0,C 180,E1 -17341.287,E2 -17341.287} C_VEL
LIN {X 0,Y 288.41,Z 212.297,A -85,B 0,C 180,E1 -17342.16,E2 -17342.16} C_VEL
LIN {X 0,Y 292.224,Z 235.213,A -85,B 0,C 180,E1 -17343.173,E2 -17343.173} C_VEL
LIN {X 0,Y 290.326,Z 300.742,A -85,B 0,C 180,E1 -17344.793,E2 -17344.793} C_VEL
LIN {X 0,Y 289.273,Z 314.648,A -85,B 0,C 180,E1 -17345.414,E2 -17345.414} C_VEL
LIN {X 0,Y 287.929,Z 327.084,A -85,B 0,C 180,E1 -17346.25,E2 -17346.25} C_VEL
LIN {X 0,Y 286.521,Z 338.175,A -85,B 0,C 180,E1 -17347.274,E2 -17347.274} C_VEL
LIN {X 0,Y 284.738,Z 349.729,A -85,B 0,C 180,E1 -17348.65,E2 -17348.65} C_VEL
LIN {X 0,Y 282.878,Z 360.131,A -85,B 0,C 180,E1 -17350.214,E2 -17350.214} C_VEL
LIN {X 0,Y 281.351,Z 368.838,A -85,B 0,C 180,E1 -17351.848,E2 -17351.848} C_VEL
LIN {X 0,Y 279.597,Z 377.851,A -85,B 0,C 180,E1 -17353.948,E2 -17353.948} C_VEL
LIN {X 0,Y 278.02,Z 385.254,A -85,B 0,C 180,E1 -17356.104,E2 -17356.104} C_VEL
LIN {X 0,Y 276.938,Z 391.2,A -85,B 0,C 180,E1 -17358.286,E2 -17358.286} C_VEL
LIN {X 0,Y 276.104,Z 395.896,A -85,B 0,C 180,E1 -17360.476,E2 -17360.476} C_VEL
LIN {X 0,Y 275.6,Z 399.483,A -85,B 0,C 180,E1 -17362.674,E2 -17362.674} C_VEL
LIN {X 0,Y 275.322,Z 401.775,A -85,B 0,C 180,E1 -17364.583,E2 -17364.583} C_VEL
LIN {X 0,Y 275.223,Z 403.707,A -85,B 0,C 180,E1 -17367.072,E2 -17367.072} C_VEL
LIN {X 0,Y 275.224,Z 404.31,A -85,B 0,C 180,E1 -17368.536,E2 -17368.536} C_VEL
LIN {X 0,Y 275.219,Z 404.521,A -85,B 0,C 180,E1 -17369.999,E2 -17369.999} C_VEL
LIN {X 0,Y 275.224,Z 404.302,A -85,B 0,C 180,E1 -17371.463,E2 -17371.463} C_VEL
LIN {X 0,Y 275.223,Z 403.693,A -85,B 0,C 180,E1 -17372.927,E2 -17372.927} C_VEL
LIN {X 0,Y 275.387,Z 401.61,A -85,B 0,C 180,E1 -17375.557,E2 -17375.557} C_VEL
LIN {X 0,Y 275.74,Z 398.376,A -85,B 0,C 180,E1 -17378.058,E2 -17378.058} C_VEL
LIN {X 0,Y 276.318,Z 394.411,A -85,B 0,C 180,E1 -17380.255,E2 -17380.255} C_VEL
LIN {X 0,Y 277.432,Z 388.315,A -85,B 0,C 180,E1 -17382.805,E2 -17382.805} C_VEL
LIN {X 0,Y 278.795,Z 381.655,A -85,B 0,C 180,E1 -17384.973,E2 -17384.973} C_VEL
LIN {X 0,Y 280.41,Z 373.389,A -85,B 0,C 180,E1 -17387.126,E2 -17387.126} C_VEL
LIN {X 0,Y 281.987,Z 364.91,A -85,B 0,C 180,E1 -17388.904,E2 -17388.904} C_VEL
LIN {X 0,Y 283.835,Z 354.431,A -85,B 0,C 180,E1 -17390.66,E2 -17390.66} C_VEL
LIN {X 0,Y 285.79,Z 342.632,A -85,B 0,C 180,E1 -17392.214,E2 -17392.214} C_VEL
LIN {X 0,Y 287.455,Z 330.745,A -85,B 0,C 180,E1 -17393.408,E2 -17393.408} C_VEL
LIN {X 0,Y 288.872,Z 318.369,A -85,B 0,C 180,E1 -17394.334,E2 -17394.334} C_VEL
LIN {X 0,Y 289.985,Z 305.623,A -85,B 0,C 180,E1 -17394.998,E2 -17394.998} C_VEL
LIN {X 0,Y 290.623,Z 292.148,A -85,B 0,C 180,E1 -17395.418,E2 -17395.418} C_VEL
LIN {X 0,Y 292.132,Z 234.719,A -85,B 0,C 180,E1 -17396.816,E2 -17396.816} C_VEL
LIN {X 0,Y 288.205,Z 211.589,A -85,B 0,C 180,E1 -17397.846,E2 -17397.846} C_VEL
LIN {X 0,Y 281.251,Z 195.052,A -85,B 0,C 180,E1 -17399.066,E2 -17399.066} C_VEL
LIN {X 0,Y 280.334,Z 192.598,A -85,B 0,C 180,E1 -17399.313,E2 -17399.313} C_VEL
LIN {X 0,Y 278.237,Z 183.2,A -85,B 0,C 180,E1 -17402.81,E2 -17402.81} C_VEL
LIN {X 0,Y 277.281,Z 178.972,A -85,B 0,C 180,E1 -17404.575,E2 -17404.575} C_VEL
LIN {X 0,Y 277.252,Z 178.922,A -85,B 0,C 180,E1 -17408.204,E2 -17408.204} C_VEL
LIN {X 0,Y 277.21,Z 178.947,A -85,B 0,C 180,E1 -17412.674,E2 -17412.674} C_VEL
LIN {X 0,Y 277.204,Z 178.944,A -85,B 0,C 180,E1 -17416.801,E2 -17416.801} C_VEL
LIN {X 0,Y 277.228,Z 178.939,A -85,B 0,C 180,E1 -17420.671,E2 -17420.671} C_VEL
LIN {X 0,Y 277.277,Z 178.906,A -85,B 0,C 180,E1 -17424.34,E2 -17424.34} C_VEL
LIN {X 0,Y 277.236,Z 178.951,A -85,B 0,C 180,E1 -17427.835,E2 -17427.835} C_VEL
LIN {X 0,Y 277.26,Z 178.938,A -85,B 0,C 180,E1 -17431.209,E2 -17431.209} C_VEL
LIN {X 0,Y 277.3,Z 178.938,A -85,B 0,C 180,E1 -17434.478,E2 -17434.478} C_VEL
LIN {X 0,Y 277.258,Z 178.945,A -85,B 0,C 180,E1 -17437.652,E2 -17437.652} C_VEL
LIN {X 0,Y 277.319,Z 178.93,A -85,B 0,C 180,E1 -17440.764,E2 -17440.764} C_VEL
LIN {X 0,Y 277.401,Z 178.93,A -85,B 0,C 180,E1 -17445.324,E2 -17445.324} C_VEL
LIN {X 0,Y 277.498,Z 178.908,A -85,B 0,C 180,E1 -17449.788,E2 -17449.788} C_VEL
LIN {X 0,Y 277.639,Z 178.899,A -85,B 0,C 180,E1 -17452.729,E2 -17452.729} C_VEL
LIN {X 0,Y 277.811,Z 178.881,A -85,B 0,C 180,E1 -17458.55,E2 -17458.55} C_VEL
LIN {X 0,Y 277.811,Z 178.864,A -85,B 0,C 180,E1 -17461.45,E2 -17461.45} C_VEL
LIN {X 0,Y 277.643,Z 178.894,A -85,B 0,C 180,E1 -17467.271,E2 -17467.271} C_VEL
LIN {X 0,Y 277.498,Z 178.901,A -85,B 0,C 180,E1 -17470.212,E2 -17470.212} C_VEL
LIN {X 0,Y 277.419,Z 178.914,A -85,B 0,C 180,E1 -17474.675,E2 -17474.675} C_VEL
LIN {X 0,Y 277.337,Z 178.938,A -85,B 0,C 180,E1 -17479.235,E2 -17479.235} C_VEL
LIN {X 0,Y 277.311,Z 178.939,A -85,B 0,C 180,E1 -17484.171,E2 -17484.171} C_VEL
LIN {X 0,Y 277.317,Z 178.928,A -85,B 0,C 180,E1 -17487.506,E2 -17487.506} C_VEL
LIN {X 0,Y 277.265,Z 178.948,A -85,B 0,C 180,E1 -17490.482,E2 -17490.482} C_VEL
LIN {X 0,Y 277.24,Z 178.91,A -85,B 0,C 180,E1 -17493.897,E2 -17493.897} C_VEL
LIN {X 0,Y 277.261,Z 178.925,A -85,B 0,C 180,E1 -17497.471,E2 -17497.471} C_VEL
LIN {X 0,Y 277.204,Z 178.943,A -85,B 0,C 180,E1 -17501.238,E2 -17501.238} C_VEL
LIN {X 0,Y 277.196,Z 178.938,A -85,B 0,C 180,E1 -17505.228,E2 -17505.228} C_VEL
LIN {X 0,Y 277.218,Z 178.926,A -85,B 0,C 180,E1 -17509.514,E2 -17509.514} C_VEL
LIN {X 0,Y 277.262,Z 178.947,A -85,B 0,C 180,E1 -17512.532,E2 -17512.532} C_VEL
LIN {X 0,Y 277.244,Z 178.936,A -85,B 0,C 180,E1 -17516.106,E2 -17516.106} C_VEL
LIN {X 0,Y 277.316,Z 179.201,A -85,B 0,C 180,E1 -17517.124,E2 -17517.124} C_VEL
LIN {X 0,Y 279.456,Z 188.237,A -85,B 0,C 180,E1 -17520.637,E2 -17520.637} C_VEL
LIN {X 0,Y 281.695,Z 193.433,A -85,B 0,C 180,E1 -17521.111,E2 -17521.111} C_VEL
LIN {X 0,Y 288.145,Z 208.772,A -85,B 0,C 180,E1 -17522.243,E2 -17522.243} C_VEL
LIN {X 0,Y 290.092,Z 214.183,A -85,B 0,C 180,E1 -17522.594,E2 -17522.594} C_VEL
LIN {X 0,Y 292.312,Z 227.602,A -85,B 0,C 180,E1 -17523.183,E2 -17523.183} C_VEL
LIN {X 0,Y 290.389,Z 296.39,A -85,B 0,C 180,E1 -17524.895,E2 -17524.895} C_VEL
LIN {X 0,Y 289.342,Z 310.129,A -85,B 0,C 180,E1 -17525.517,E2 -17525.517} C_VEL
LIN {X 0,Y 288.19,Z 322.461,A -85,B 0,C 180,E1 -17526.37,E2 -17526.37} C_VEL
LIN {X 0,Y 286.622,Z 334.289,A -85,B 0,C 180,E1 -17527.474,E2 -17527.474} C_VEL
LIN {X 0,Y 284.816,Z 345.651,A -85,B 0,C 180,E1 -17528.847,E2 -17528.847} C_VEL
LIN {X 0,Y 283.241,Z 355.151,A -85,B 0,C 180,E1 -17530.298,E2 -17530.298} C_VEL
LIN {X 0,Y 281.81,Z 363.484,A -85,B 0,C 180,E1 -17531.858,E2 -17531.858} C_VEL
LIN {X 0,Y 280.262,Z 371.271,A -85,B 0,C 180,E1 -17533.615,E2 -17533.615} C_VEL
LIN {X 0,Y 278.602,Z 378.978,A -85,B 0,C 180,E1 -17535.763,E2 -17535.763} C_VEL
LIN {X 0,Y 277.254,Z 386.055,A -85,B 0,C 180,E1 -17538.301,E2 -17538.301} C_VEL
LIN {X 0,Y 276.368,Z 390.769,A -85,B 0,C 180,E1 -17540.487,E2 -17540.487} C_VEL
LIN {X 0,Y 275.776,Z 394.377,A -85,B 0,C 180,E1 -17542.68,E2 -17542.68} C_VEL
LIN {X 0,Y 275.551,Z 396.241,A -85,B 0,C 180,E1 -17544.145,E2 -17544.145} C_VEL
LIN {X 0,Y 275.367,Z 397.643,A -85,B 0,C 180,E1 -17545.609,E2 -17545.609} C_VEL
LIN {X 0,Y 275.289,Z 398.64,A -85,B 0,C 180,E1 -17547.074,E2 -17547.074} C_VEL
LIN {X 0,Y 275.24,Z 399.254,A -85,B 0,C 180,E1 -17548.538,E2 -17548.538} C_VEL
LIN {X 0,Y 275.221,Z 399.486,A -85,B 0,C 180,E1 -17550.001,E2 -17550.001} C_VEL
LIN {X 0,Y 275.24,Z 399.292,A -85,B 0,C 180,E1 -17551.464,E2 -17551.464} C_VEL
LIN {X 0,Y 275.287,Z 398.703,A -85,B 0,C 180,E1 -17552.927,E2 -17552.927} C_VEL
LIN {X 0,Y 275.532,Z 396.367,A -85,B 0,C 180,E1 -17555.856,E2 -17555.856} C_VEL
LIN {X 0,Y 275.949,Z 393.485,A -85,B 0,C 180,E1 -17558.053,E2 -17558.053} C_VEL
LIN {X 0,Y 276.593,Z 389.579,A -85,B 0,C 180,E1 -17560.246,E2 -17560.246} C_VEL
LIN {X 0,Y 277.553,Z 384.541,A -85,B 0,C 180,E1 -17562.429,E2 -17562.429} C_VEL
LIN {X 0,Y 278.787,Z 378.199,A -85,B 0,C 180,E1 -17564.602,E2 -17564.602} C_VEL
LIN {X 0,Y 280.485,Z 370.264,A -85,B 0,C 180,E1 -17566.748,E2 -17566.748} C_VEL
LIN {X 0,Y 282.023,Z 362.002,A -85,B 0,C 180,E1 -17568.563,E2 -17568.563} C_VEL
LIN {X 0,Y 283.679,Z 352.311,A -85,B 0,C 180,E1 -17570.294,E2 -17570.294} C_VEL
LIN {X 0,Y 285.627,Z 341.207,A -85,B 0,C 180,E1 -17571.849,E2 -17571.849} C_VEL
LIN {X 0,Y 287.25,Z 330.323,A -85,B 0,C 180,E1 -17573.046,E2 -17573.046} C_VEL
LIN {X 0,Y 288.659,Z 318.298,A -85,B 0,C 180,E1 -17574.068,E2 -17574.068} C_VEL
LIN {X 0,Y 289.754,Z 305.941,A -85,B 0,C 180,E1 -17574.829,E2 -17574.829} C_VEL
LIN {X 0,Y 290.556,Z 293.131,A -85,B 0,C 180,E1 -17575.33,E2 -17575.33} C_VEL
LIN {X 0,Y 292.313,Z 226.447,A -85,B 0,C 180,E1 -17576.971,E2 -17576.971} C_VEL
LIN {X 0,Y 289.643,Z 212.564,A -85,B 0,C 180,E1 -17577.621,E2 -17577.621} C_VEL
LIN {X 0,Y 282.102,Z 194.296,A -85,B 0,C 180,E1 -17578.946,E2 -17578.946} C_VEL
LIN {X 0,Y 279.495,Z 188.294,A -85,B 0,C 180,E1 -17579.475,E2 -17579.475} C_VEL
LIN {X 0,Y 277.354,Z 179.496,A -85,B 0,C 180,E1 -17582.873,E2 -17582.873} C_VEL
LIN {X 0,Y 277.256,Z 178.963,A -85,B 0,C 180,E1 -17583.227,E2 -17583.227} C_VEL
LIN {X 0,Y 277.324,Z 178.925,A -85,B 0,C 180,E1 -17585.811,E2 -17585.811} C_VEL
LIN {X 0,Y 277.236,Z 178.924,A -85,B 0,C 180,E1 -17589.327,E2 -17589.327} C_VEL
LIN {X 0,Y 277.209,Z 178.955,A -85,B 0,C 180,E1 -17593.198,E2 -17593.198} C_VEL
LIN {X 0,Y 277.214,Z 178.92,A -85,B 0,C 180,E1 -17597.325,E2 -17597.325} C_VEL
LIN {X 0,Y 277.264,Z 178.94,A -85,B 0,C 180,E1 -17601.792,E2 -17601.792} C_VEL
LIN {X 0,Y 277.283,Z 178.897,A -85,B 0,C 180,E1 -17604.341,E2 -17604.341} C_VEL
LIN {X 0,Y 277.243,Z 178.937,A -85,B 0,C 180,E1 -17607.836,E2 -17607.836} C_VEL
LIN {X 0,Y 277.287,Z 178.938,A -85,B 0,C 180,E1 -17611.212,E2 -17611.212} C_VEL
LIN {X 0,Y 277.306,Z 178.943,A -85,B 0,C 180,E1 -17614.479,E2 -17614.479} C_VEL
LIN {X 0,Y 277.252,Z 178.936,A -85,B 0,C 180,E1 -17617.085,E2 -17617.085} C_VEL
LIN {X 0,Y 276.594,Z 179.019,A -85,B 0,C 180,E1 -17618.297,E2 -17618.297} C_VEL
LIN {X 0,Y 273.77,Z 179.383,A -85,B 0,C 180,E1 -17620.274,E2 -17620.274} C_VEL
LIN {X 0,Y 271.391,Z 179.677,A -85,B 0,C 180,E1 -17621.88,E2 -17621.88} C_VEL
LIN {X 0,Y 270.4,Z 179.791,A -85,B 0,C 180,E1 -17623.123,E2 -17623.123} C_VEL
LIN {X 0,Y 270.336,Z 179.794,A -85,B 0,C 180,E1 -17623.545,E2 -17623.545} C_VEL
LIN {X 0,Y 270.354,Z 179.805,A -85,B 0,C 180,E1 -17626.47,E2 -17626.47} C_VEL
LIN {X 0,Y 270.574,Z 179.759,A -85,B 0,C 180,E1 -17631.034,E2 -17631.034} C_VEL
LIN {X 0,Y 270.537,Z 179.785,A -85,B 0,C 180,E1 -17634.035,E2 -17634.035} C_VEL
LIN {X 0,Y 270.782,Z 179.738,A -85,B 0,C 180,E1 -17638.513,E2 -17638.513} C_VEL
LIN {X 0,Y 270.781,Z 179.756,A -85,B 0,C 180,E1 -17641.487,E2 -17641.487} C_VEL
LIN {X 0,Y 270.58,Z 179.78,A -85,B 0,C 180,E1 -17647.462,E2 -17647.462} C_VEL
LIN {X 0,Y 270.385,Z 179.79,A -85,B 0,C 180,E1 -17650.483,E2 -17650.483} C_VEL
LIN {X 0,Y 270.374,Z 179.808,A -85,B 0,C 180,E1 -17655.066,E2 -17655.066} C_VEL
LIN {X 0,Y 270.276,Z 179.814,A -85,B 0,C 180,E1 -17659.757,E2 -17659.757} C_VEL
LIN {X 0,Y 270.235,Z 179.81,A -85,B 0,C 180,E1 -17664.589,E2 -17664.589} C_VEL
LIN {X 0,Y 270.268,Z 179.815,A -85,B 0,C 180,E1 -17667.909,E2 -17667.909} C_VEL
LIN {X 0,Y 270.182,Z 179.83,A -85,B 0,C 180,E1 -17671.349,E2 -17671.349} C_VEL
LIN {X 0,Y 270.2,Z 179.795,A -85,B 0,C 180,E1 -17674.906,E2 -17674.906} C_VEL
LIN {X 0,Y 270.196,Z 179.805,A -85,B 0,C 180,E1 -17678.711,E2 -17678.711} C_VEL
LIN {X 0,Y 270.17,Z 179.821,A -85,B 0,C 180,E1 -17682.559,E2 -17682.559} C_VEL
LIN {X 0,Y 270.164,Z 179.824,A -85,B 0,C 180,E1 -17686.751,E2 -17686.751} C_VEL
LIN {X 0,Y 270.173,Z 179.826,A -85,B 0,C 180,E1 -17689.434,E2 -17689.434} C_VEL
LIN {X 0,Y 270.239,Z 179.819,A -85,B 0,C 180,E1 -17693.727,E2 -17693.727} C_VEL
LIN {X 0,Y 270.265,Z 180.082,A -85,B 0,C 180,E1 -17694.877,E2 -17694.877} C_VEL
LIN {X 0,Y 271.985,Z 187.438,A -85,B 0,C 180,E1 -17697.885,E2 -17697.885} C_VEL
LIN {X 0,Y 273.147,Z 192.68,A -85,B 0,C 180,E1 -17699.826,E2 -17699.826} C_VEL
LIN {X 0,Y 279.732,Z 207.988,A -85,B 0,C 180,E1 -17701.095,E2 -17701.095} C_VEL
LIN {X 0,Y 282.465,Z 215.337,A -85,B 0,C 180,E1 -17701.608,E2 -17701.608} C_VEL
LIN {X 0,Y 285.896,Z 236.004,A -85,B 0,C 180,E1 -17702.553,E2 -17702.553} C_VEL
LIN {X 0,Y 283.935,Z 300.691,A -85,B 0,C 180,E1 -17704.184,E2 -17704.184} C_VEL
LIN {X 0,Y 282.843,Z 314.592,A -85,B 0,C 180,E1 -17704.817,E2 -17704.817} C_VEL
LIN {X 0,Y 281.465,Z 327.026,A -85,B 0,C 180,E1 -17705.67,E2 -17705.67} C_VEL
LIN {X 0,Y 279.992,Z 338.115,A -85,B 0,C 180,E1 -17706.713,E2 -17706.713} C_VEL
LIN {X 0,Y 278.116,Z 349.668,A -85,B 0,C 180,E1 -17708.116,E2 -17708.116} C_VEL
LIN {X 0,Y 276.192,Z 360.07,A -85,B 0,C 180,E1 -17709.714,E2 -17709.714} C_VEL
LIN {X 0,Y 274.457,Z 369.453,A -85,B 0,C 180,E1 -17711.531,E2 -17711.531} C_VEL
LIN {X 0,Y 272.757,Z 377.787,A -85,B 0,C 180,E1 -17713.535,E2 -17713.535} C_VEL
LIN {X 0,Y 271.121,Z 385.191,A -85,B 0,C 180,E1 -17715.743,E2 -17715.743} C_VEL
LIN {X 0,Y 269.96,Z 391.136,A -85,B 0,C 180,E1 -17717.979,E2 -17717.979} C_VEL
LIN {X 0,Y 269.071,Z 395.832,A -85,B 0,C 180,E1 -17720.225,E2 -17720.225} C_VEL
LIN {X 0,Y 268.537,Z 399.418,A -85,B 0,C 180,E1 -17722.48,E2 -17722.48} C_VEL
LIN {X 0,Y 268.215,Z 401.954,A -85,B 0,C 180,E1 -17724.691,E2 -17724.691} C_VEL
LIN {X 0,Y 268.12,Z 403.642,A -85,B 0,C 180,E1 -17726.994,E2 -17726.994} C_VEL
LIN {X 0,Y 268.13,Z 404.245,A -85,B 0,C 180,E1 -17728.497,E2 -17728.497} C_VEL
LIN {X 0,Y 268.146,Z 404.457,A -85,B 0,C 180,E1 -17729.999,E2 -17729.999} C_VEL
LIN {X 0,Y 268.13,Z 404.236,A -85,B 0,C 180,E1 -17731.501,E2 -17731.501} C_VEL
LIN {X 0,Y 268.121,Z 403.628,A -85,B 0,C 180,E1 -17733.004,E2 -17733.004} C_VEL
LIN {X 0,Y 268.294,Z 401.755,A -85,B 0,C 180,E1 -17735.486,E2 -17735.486} C_VEL
LIN {X 0,Y 268.698,Z 398.31,A -85,B 0,C 180,E1 -17738.27,E2 -17738.27} C_VEL
LIN {X 0,Y 269.312,Z 394.345,A -85,B 0,C 180,E1 -17740.525,E2 -17740.525} C_VEL
LIN {X 0,Y 270.467,Z 388.248,A -85,B 0,C 180,E1 -17743.141,E2 -17743.141} C_VEL
LIN {X 0,Y 271.907,Z 381.588,A -85,B 0,C 180,E1 -17745.362,E2 -17745.362} C_VEL
LIN {X 0,Y 273.618,Z 373.322,A -85,B 0,C 180,E1 -17747.565,E2 -17747.565} C_VEL
LIN {X 0,Y 275.26,Z 364.842,A -85,B 0,C 180,E1 -17749.384,E2 -17749.384} C_VEL
LIN {X 0,Y 277.206,Z 354.363,A -85,B 0,C 180,E1 -17751.178,E2 -17751.178} C_VEL
LIN {X 0,Y 279.215,Z 342.563,A -85,B 0,C 180,E1 -17752.767,E2 -17752.767} C_VEL
LIN {X 0,Y 280.966,Z 330.674,A -85,B 0,C 180,E1 -17753.982,E2 -17753.982} C_VEL
LIN {X 0,Y 282.395,Z 318.296,A -85,B 0,C 180,E1 -17754.93,E2 -17754.93} C_VEL
LIN {X 0,Y 283.586,Z 305.546,A -85,B 0,C 180,E1 -17755.602,E2 -17755.602} C_VEL
LIN {X 0,Y 284.231,Z 292.062,A -85,B 0,C 180,E1 -17756.032,E2 -17756.032} C_VEL
LIN {X 0,Y 285.735,Z 235.268,A -85,B 0,C 180,E1 -17757.449,E2 -17757.449} C_VEL
LIN {X 0,Y 282.107,Z 214.074,A -85,B 0,C 180,E1 -17758.43,E2 -17758.43} C_VEL
LIN {X 0,Y 275.623,Z 198.424,A -85,B 0,C 180,E1 -17759.617,E2 -17759.617} C_VEL
LIN {X 0,Y 273.151,Z 192.651,A -85,B 0,C 180,E1 -17760.136,E2 -17760.136} C_VEL
LIN {X 0,Y 270.946,Z 182.888,A -85,B 0,C 180,E1 -17763.897,E2 -17763.897} C_VEL
LIN {X 0,Y 270.251,Z 179.834,A -85,B 0,C 180,E1 -17765.266,E2 -17765.266} C_VEL
LIN {X 0,Y 270.194,Z 179.801,A -85,B 0,C 180,E1 -17768.709,E2 -17768.709} C_VEL
LIN {X 0,Y 270.167,Z 179.824,A -85,B 0,C 180,E1 -17772.557,E2 -17772.557} C_VEL
LIN {X 0,Y 270.159,Z 179.821,A -85,B 0,C 180,E1 -17776.75,E2 -17776.75} C_VEL
LIN {X 0,Y 270.168,Z 179.831,A -85,B 0,C 180,E1 -17779.433,E2 -17779.433} C_VEL
LIN {X 0,Y 270.219,Z 179.779,A -85,B 0,C 180,E1 -17783.73,E2 -17783.73} C_VEL
LIN {X 0,Y 270.196,Z 179.824,A -85,B 0,C 180,E1 -17786.891,E2 -17786.891} C_VEL
LIN {X 0,Y 270.188,Z 179.816,A -85,B 0,C 180,E1 -17790.382,E2 -17790.382} C_VEL
LIN {X 0,Y 270.252,Z 179.82,A -85,B 0,C 180,E1 -17793.763,E2 -17793.763} C_VEL
LIN {X 0,Y 270.2,Z 179.816,A -85,B 0,C 180,E1 -17797.036,E2 -17797.036} C_VEL
LIN {X 0,Y 270.27,Z 179.814,A -85,B 0,C 180,E1 -17800.242,E2 -17800.242} C_VEL
LIN {X 0,Y 270.368,Z 179.808,A -85,B 0,C 180,E1 -17804.933,E2 -17804.933} C_VEL
LIN {X 0,Y 270.433,Z 179.784,A -85,B 0,C 180,E1 -17809.519,E2 -17809.519} C_VEL
LIN {X 0,Y 270.598,Z 179.777,A -85,B 0,C 180,E1 -17812.538,E2 -17812.538} C_VEL
LIN {X 0,Y 270.777,Z 179.757,A -85,B 0,C 180,E1 -17818.513,E2 -17818.513} C_VEL
LIN {X 0,Y 270.776,Z 179.739,A -85,B 0,C 180,E1 -17821.487,E2 -17821.487} C_VEL
LIN {X 0,Y 270.601,Z 179.771,A -85,B 0,C 180,E1 -17827.462,E2 -17827.462} C_VEL
LIN {X 0,Y 270.433,Z 179.783,A -85,B 0,C 180,E1 -17830.481,E2 -17830.481} C_VEL
LIN {X 0,Y 270.388,Z 179.787,A -85,B 0,C 180,E1 -17835.066,E2 -17835.066} C_VEL
LIN {X 0,Y 270.294,Z 179.816,A -85,B 0,C 180,E1 -17839.756,E2 -17839.756} C_VEL
LIN {X 0,Y 270.267,Z 179.821,A -85,B 0,C 180,E1 -17844.586,E2 -17844.586} C_VEL
LIN {X 0,Y 270.265,Z 179.806,A -85,B 0,C 180,E1 -17847.91,E2 -17847.91} C_VEL
LIN {X 0,Y 270.178,Z 179.829,A -85,B 0,C 180,E1 -17851.349,E2 -17851.349} C_VEL
LIN {X 0,Y 270.195,Z 179.778,A -85,B 0,C 180,E1 -17854.907,E2 -17854.907} C_VEL
LIN {X 0,Y 270.192,Z 179.825,A -85,B 0,C 180,E1 -17858.712,E2 -17858.712} C_VEL
LIN {X 0,Y 270.166,Z 179.8,A -85,B 0,C 180,E1 -17862.56,E2 -17862.56} C_VEL
LIN {X 0,Y 270.161,Z 179.833,A -85,B 0,C 180,E1 -17866.752,E2 -17866.752} C_VEL
LIN {X 0,Y 270.194,Z 179.805,A -85,B 0,C 180,E1 -17871.291,E2 -17871.291} C_VEL
LIN {X 0,Y 270.199,Z 179.809,A -85,B 0,C 180,E1 -17875.096,E2 -17875.096} C_VEL
LIN {X 0,Y 270.213,Z 179.903,A -85,B 0,C 180,E1 -17876.335,E2 -17876.335} C_VEL
LIN {X 0,Y 272.13,Z 187.98,A -85,B 0,C 180,E1 -17879.683,E2 -17879.683} C_VEL
LIN {X 0,Y 272.556,Z 189.35,A -85,B 0,C 180,E1 -17879.906,E2 -17879.906} C_VEL
LIN {X 0,Y 278.866,Z 203.2,A -85,B 0,C 180,E1 -17881.071,E2 -17881.071} C_VEL
LIN {X 0,Y 284.012,Z 216.461,A -85,B 0,C 180,E1 -17882.018,E2 -17882.018} C_VEL
LIN {X 0,Y 285.998,Z 228.432,A -85,B 0,C 180,E1 -17882.563,E2 -17882.563} C_VEL
LIN {X 0,Y 283.995,Z 296.47,A -85,B 0,C 180,E1 -17884.29,E2 -17884.29} C_VEL
LIN {X 0,Y 282.904,Z 310.204,A -85,B 0,C 180,E1 -17884.922,E2 -17884.922} C_VEL
LIN {X 0,Y 281.713,Z 322.533,A -85,B 0,C 180,E1 -17885.792,E2 -17885.792} C_VEL
LIN {X 0,Y 280.07,Z 334.359,A -85,B 0,C 180,E1 -17886.917,E2 -17886.917} C_VEL
LIN {X 0,Y 278.194,Z 345.72,A -85,B 0,C 180,E1 -17888.318,E2 -17888.318} C_VEL
LIN {X 0,Y 276.541,Z 355.22,A -85,B 0,C 180,E1 -17889.8,E2 -17889.8} C_VEL
LIN {X 0,Y 274.989,Z 363.865,A -85,B 0,C 180,E1 -17891.46,E2 -17891.46} C_VEL
LIN {X 0,Y 273.146,Z 372.729,A -85,B 0,C 180,E1 -17893.56,E2 -17893.56} C_VEL
LIN {X 0,Y 271.478,Z 380.159,A -85,B 0,C 180,E1 -17895.764,E2 -17895.764} C_VEL
LIN {X 0,Y 270.272,Z 386.122,A -85,B 0,C 180,E1 -17897.994,E2 -17897.994} C_VEL
LIN {X 0,Y 269.363,Z 390.835,A -85,B 0,C 180,E1 -17900.237,E2 -17900.237} C_VEL
LIN {X 0,Y 268.731,Z 394.443,A -85,B 0,C 180,E1 -17902.487,E2 -17902.487} C_VEL
LIN {X 0,Y 268.482,Z 396.436,A -85,B 0,C 180,E1 -17904.113,E2 -17904.113} C_VEL
LIN {X 0,Y 268.205,Z 398.706,A -85,B 0,C 180,E1 -17906.997,E2 -17906.997} C_VEL
LIN {X 0,Y 268.147,Z 399.319,A -85,B 0,C 180,E1 -17908.499,E2 -17908.499} C_VEL
LIN {X 0,Y 268.148,Z 399.55,A -85,B 0,C 180,E1 -17910.001,E2 -17910.001} C_VEL
LIN {X 0,Y 268.147,Z 399.357,A -85,B 0,C 180,E1 -17911.502,E2 -17911.502} C_VEL
LIN {X 0,Y 268.203,Z 398.768,A -85,B 0,C 180,E1 -17913.005,E2 -17913.005} C_VEL
LIN {X 0,Y 268.462,Z 396.431,A -85,B 0,C 180,E1 -17916.011,E2 -17916.011} C_VEL
LIN {X 0,Y 268.923,Z 393.549,A -85,B 0,C 180,E1 -17918.265,E2 -17918.265} C_VEL
LIN {X 0,Y 269.588,Z 389.643,A -85,B 0,C 180,E1 -17920.515,E2 -17920.515} C_VEL
LIN {X 0,Y 270.608,Z 384.605,A -85,B 0,C 180,E1 -17922.754,E2 -17922.754} C_VEL
LIN {X 0,Y 271.918,Z 378.262,A -85,B 0,C 180,E1 -17924.979,E2 -17924.979} C_VEL
LIN {X 0,Y 273.691,Z 370.326,A -85,B 0,C 180,E1 -17927.176,E2 -17927.176} C_VEL
LIN {X 0,Y 275.538,Z 360.714,A -85,B 0,C 180,E1 -17929.31,E2 -17929.31} C_VEL
LIN {X 0,Y 277.241,Z 351.273,A -85,B 0,C 180,E1 -17930.982,E2 -17930.982} C_VEL
LIN {X 0,Y 279.265,Z 339.843,A -85,B 0,C 180,E1 -17932.568,E2 -17932.568} C_VEL
LIN {X 0,Y 280.93,Z 328.618,A -85,B 0,C 180,E1 -17933.791,E2 -17933.791} C_VEL
LIN {X 0,Y 282.439,Z 315.958,A -85,B 0,C 180,E1 -17934.829,E2 -17934.829} C_VEL
LIN {X 0,Y 283.584,Z 303.26,A -85,B 0,C 180,E1 -17935.555,E2 -17935.555} C_VEL
LIN {X 0,Y 284.286,Z 290.166,A -85,B 0,C 180,E1 -17936.028,E2 -17936.028} C_VEL
LIN {X 0,Y 285.965,Z 227.221,A -85,B 0,C 180,E1 -17937.6,E2 -17937.6} C_VEL
LIN {X 0,Y 283.684,Z 215.257,A -85,B 0,C 180,E1 -17938.178,E2 -17938.178} C_VEL
LIN {X 0,Y 276.251,Z 197.196,A -85,B 0,C 180,E1 -17939.536,E2 -17939.536} C_VEL
LIN {X 0,Y 272.302,Z 188.475,A -85,B 0,C 180,E1 -17940.317,E2 -17940.317} C_VEL
LIN {X 0,Y 270.614,Z 181.512,A -85,B 0,C 180,E1 -17943.051,E2 -17943.051} C_VEL
LIN {X 0,Y 270.226,Z 179.846,A -85,B 0,C 180,E1 -17943.871,E2 -17943.871} C_VEL
LIN {X 0,Y 270.237,Z 179.82,A -85,B 0,C 180,E1 -17946.738,E2 -17946.738} C_VEL
LIN {X 0,Y 270.169,Z 179.806,A -85,B 0,C 180,E1 -17951.028,E2 -17951.028} C_VEL
LIN {X 0,Y 270.152,Z 179.821,A -85,B 0,C 180,E1 -17954.62,E2 -17954.62} C_VEL
LIN {X 0,Y 270.171,Z 179.798,A -85,B 0,C 180,E1 -17957.441,E2 -17957.441} C_VEL
LIN {X 0,Y 270.206,Z 179.825,A -85,B 0,C 180,E1 -17961.374,E2 -17961.374} C_VEL
LIN {X 0,Y 270.2,Z 179.776,A -85,B 0,C 180,E1 -17965.094,E2 -17965.094} C_VEL
LIN {X 0,Y 270.199,Z 179.826,A -85,B 0,C 180,E1 -17969.13,E2 -17969.13} C_VEL
LIN {X 0,Y 270.263,Z 179.806,A -85,B 0,C 180,E1 -17972.145,E2 -17972.145} C_VEL
LIN {X 0,Y 270.235,Z 179.825,A -85,B 0,C 180,E1 -17975.537,E2 -17975.537} C_VEL
LIN {X 0,Y 270.298,Z 179.815,A -85,B 0,C 180,E1 -17980.244,E2 -17980.244} C_VEL
LIN {X 0,Y 270.336,Z 179.794,A -85,B 0,C 180,E1 -17983.545,E2 -17983.545} C_VEL
LIN {X 0,Y 269.697,Z 179.873,A -85,B 0,C 180,E1 -17984.789,E2 -17984.789} C_VEL
LIN {X 0,Y 266.831,Z 180.244,A -85,B 0,C 180,E1 -17986.816,E2 -17986.816} C_VEL
LIN {X 0,Y 264.435,Z 180.541,A -85,B 0,C 180,E1 -17988.465,E2 -17988.465} C_VEL
LIN {X 0,Y 263.488,Z 180.646,A -85,B 0,C 180,E1 -17989.743,E2 -17989.743} C_VEL
LIN {X 0,Y 263.457,Z 180.646,A -85,B 0,C 180,E1 -17990.175,E2 -17990.175} C_VEL
LIN {X 0,Y 263.569,Z 180.642,A -85,B 0,C 180,E1 -17992.338,E2 -17992.338} C_VEL
LIN {X 0,Y 263.747,Z 180.614,A -85,B 0,C 180,E1 -17998.473,E2 -17998.473} C_VEL
LIN {X 0,Y 263.746,Z 180.632,A -85,B 0,C 180,E1 -18001.527,E2 -18001.527} C_VEL
LIN {X 0,Y 263.54,Z 180.659,A -85,B 0,C 180,E1 -18007.663,E2 -18007.663} C_VEL
LIN {X 0,Y 263.331,Z 180.666,A -85,B 0,C 180,E1 -18010.767,E2 -18010.767} C_VEL
LIN {X 0,Y 263.32,Z 180.682,A -85,B 0,C 180,E1 -18015.48,E2 -18015.48} C_VEL
LIN {X 0,Y 263.241,Z 180.693,A -85,B 0,C 180,E1 -18020.308,E2 -18020.308} C_VEL
LIN {X 0,Y 263.19,Z 180.693,A -85,B 0,C 180,E1 -18025.293,E2 -18025.293} C_VEL
LIN {X 0,Y 263.164,Z 180.693,A -85,B 0,C 180,E1 -18028.731,E2 -18028.731} C_VEL
LIN {X 0,Y 263.131,Z 180.709,A -85,B 0,C 180,E1 -18032.289,E2 -18032.289} C_VEL
LIN {X 0,Y 263.181,Z 180.655,A -85,B 0,C 180,E1 -18036.763,E2 -18036.763} C_VEL
LIN {X 0,Y 263.123,Z 180.706,A -85,B 0,C 180,E1 -18041.594,E2 -18041.594} C_VEL
LIN {X 0,Y 263.104,Z 180.706,A -85,B 0,C 180,E1 -18046.155,E2 -18046.155} C_VEL
LIN {X 0,Y 263.105,Z 180.693,A -85,B 0,C 180,E1 -18050.128,E2 -18050.128} C_VEL
LIN {X 0,Y 263.241,Z 180.91,A -85,B 0,C 180,E1 -18054.141,E2 -18054.141} C_VEL
LIN {X 0,Y 265.078,Z 188.916,A -85,B 0,C 180,E1 -18057.529,E2 -18057.529} C_VEL
LIN {X 0,Y 265.97,Z 192.683,A -85,B 0,C 180,E1 -18058.931,E2 -18058.931} C_VEL
LIN {X 0,Y 273.515,Z 209.909,A -85,B 0,C 180,E1 -18060.431,E2 -18060.431} C_VEL
LIN {X 0,Y 276.468,Z 217.774,A -85,B 0,C 180,E1 -18061.006,E2 -18061.006} C_VEL
LIN {X 0,Y 279.604,Z 236.923,A -85,B 0,C 180,E1 -18061.908,E2 -18061.908} C_VEL
LIN {X 0,Y 277.572,Z 300.64,A -85,B 0,C 180,E1 -18063.547,E2 -18063.547} C_VEL
LIN {X 0,Y 276.454,Z 314.537,A -85,B 0,C 180,E1 -18064.192,E2 -18064.192} C_VEL
LIN {X 0,Y 274.998,Z 326.967,A -85,B 0,C 180,E1 -18065.059,E2 -18065.059} C_VEL
LIN {X 0,Y 273.229,Z 339.637,A -85,B 0,C 180,E1 -18066.303,E2 -18066.303} C_VEL
LIN {X 0,Y 271.3,Z 350.899,A -85,B 0,C 180,E1 -18067.737,E2 -18067.737} C_VEL
LIN {X 0,Y 269.319,Z 361.043,A -85,B 0,C 180,E1 -18069.372,E2 -18069.372} C_VEL
LIN {X 0,Y 267.573,Z 370.04,A -85,B 0,C 180,E1 -18071.197,E2 -18071.197} C_VEL
LIN {X 0,Y 265.655,Z 379.08,A -85,B 0,C 180,E1 -18073.477,E2 -18073.477} C_VEL
LIN {X 0,Y 263.984,Z 386.239,A -85,B 0,C 180,E1 -18075.743,E2 -18075.743} C_VEL
LIN {X 0,Y 262.634,Z 392.758,A -85,B 0,C 180,E1 -18078.422,E2 -18078.422} C_VEL
LIN {X 0,Y 261.828,Z 397.07,A -85,B 0,C 180,E1 -18080.732,E2 -18080.732} C_VEL
LIN {X 0,Y 261.482,Z 399.354,A -85,B 0,C 180,E1 -18082.276,E2 -18082.276} C_VEL
LIN {X 0,Y 261.124,Z 402.099,A -85,B 0,C 180,E1 -18084.769,E2 -18084.769} C_VEL
LIN {X 0,Y 261.021,Z 403.578,A -85,B 0,C 180,E1 -18086.913,E2 -18086.913} C_VEL
LIN {X 0,Y 261.038,Z 404.181,A -85,B 0,C 180,E1 -18088.457,E2 -18088.457} C_VEL
LIN {X 0,Y 261.074,Z 404.392,A -85,B 0,C 180,E1 -18089.999,E2 -18089.999} C_VEL
LIN {X 0,Y 261.038,Z 404.171,A -85,B 0,C 180,E1 -18091.542,E2 -18091.542} C_VEL
LIN {X 0,Y 261.087,Z 402.568,A -85,B 0,C 180,E1 -18094.631,E2 -18094.631} C_VEL
LIN {X 0,Y 261.238,Z 401.173,A -85,B 0,C 180,E1 -18096.177,E2 -18096.177} C_VEL
LIN {X 0,Y 261.643,Z 398.244,A -85,B 0,C 180,E1 -18098.495,E2 -18098.495} C_VEL
LIN {X 0,Y 262.322,Z 394.279,A -85,B 0,C 180,E1 -18100.808,E2 -18100.808} C_VEL
LIN {X 0,Y 263.527,Z 388.181,A -85,B 0,C 180,E1 -18103.494,E2 -18103.494} C_VEL
LIN {X 0,Y 265.049,Z 381.521,A -85,B 0,C 180,E1 -18105.77,E2 -18105.77} C_VEL
LIN {X 0,Y 266.85,Z 373.255,A -85,B 0,C 180,E1 -18108.025,E2 -18108.025} C_VEL
LIN {X 0,Y 268.554,Z 364.775,A -85,B 0,C 180,E1 -18109.888,E2 -18109.888} C_VEL
LIN {X 0,Y 270.577,Z 354.294,A -85,B 0,C 180,E1 -18111.722,E2 -18111.722} C_VEL
LIN {X 0,Y 272.666,Z 342.493,A -85,B 0,C 180,E1 -18113.345,E2 -18113.345} C_VEL
LIN {X 0,Y 274.513,Z 330.604,A -85,B 0,C 180,E1 -18114.583,E2 -18114.583} C_VEL
LIN {X 0,Y 275.982,Z 318.223,A -85,B 0,C 180,E1 -18115.55,E2 -18115.55} C_VEL
LIN {X 0,Y 277.222,Z 305.47,A -85,B 0,C 180,E1 -18116.234,E2 -18116.234} C_VEL
LIN {X 0,Y 277.872,Z 291.976,A -85,B 0,C 180,E1 -18116.674,E2 -18116.674} C_VEL
LIN {X 0,Y 279.453,Z 236.283,A -85,B 0,C 180,E1 -18118.089,E2 -18118.089} C_VEL
LIN {X 0,Y 276.099,Z 216.485,A -85,B 0,C 180,E1 -18119.034,E2 -18119.034} C_VEL
LIN {X 0,Y 269.056,Z 199.636,A -85,B 0,C 180,E1 -18120.376,E2 -18120.376} C_VEL
LIN {X 0,Y 265.886,Z 192.541,A -85,B 0,C 180,E1 -18121.054,E2 -18121.054} C_VEL
LIN {X 0,Y 264.001,Z 184.176,A -85,B 0,C 180,E1 -18124.386,E2 -18124.386} C_VEL
LIN {X 0,Y 263.19,Z 180.72,A -85,B 0,C 180,E1 -18125.976,E2 -18125.976} C_VEL
LIN {X 0,Y 263.101,Z 180.695,A -85,B 0,C 180,E1 -18129.871,E2 -18129.871} C_VEL
LIN {X 0,Y 263.099,Z 180.709,A -85,B 0,C 180,E1 -18133.987,E2 -18133.987} C_VEL
LIN {X 0,Y 263.119,Z 180.707,A -85,B 0,C 180,E1 -18138.405,E2 -18138.405} C_VEL
LIN {X 0,Y 263.176,Z 180.655,A -85,B 0,C 180,E1 -18143.236,E2 -18143.236} C_VEL
LIN {X 0,Y 263.126,Z 180.709,A -85,B 0,C 180,E1 -18147.711,E2 -18147.711} C_VEL
LIN {X 0,Y 263.189,Z 180.696,A -85,B 0,C 180,E1 -18151.784,E2 -18151.784} C_VEL
LIN {X 0,Y 263.193,Z 180.687,A -85,B 0,C 180,E1 -18155.212,E2 -18155.212} C_VEL
LIN {X 0,Y 263.236,Z 180.693,A -85,B 0,C 180,E1 -18159.691,E2 -18159.691} C_VEL
LIN {X 0,Y 263.315,Z 180.683,A -85,B 0,C 180,E1 -18164.52,E2 -18164.52} C_VEL
LIN {X 0,Y 263.365,Z 180.662,A -85,B 0,C 180,E1 -18169.234,E2 -18169.234} C_VEL
LIN {X 0,Y 263.56,Z 180.656,A -85,B 0,C 180,E1 -18172.338,E2 -18172.338} C_VEL
LIN {X 0,Y 263.741,Z 180.633,A -85,B 0,C 180,E1 -18178.473,E2 -18178.473} C_VEL
LIN {X 0,Y 263.741,Z 180.615,A -85,B 0,C 180,E1 -18181.527,E2 -18181.527} C_VEL
LIN {X 0,Y 263.563,Z 180.643,A -85,B 0,C 180,E1 -18187.662,E2 -18187.662} C_VEL
LIN {X 0,Y 263.365,Z 180.666,A -85,B 0,C 180,E1 -18190.766,E2 -18190.766} C_VEL
LIN {X 0,Y 263.336,Z 180.663,A -85,B 0,C 180,E1 -18195.479,E2 -18195.479} C_VEL
LIN {X 0,Y 263.256,Z 180.687,A -85,B 0,C 180,E1 -18200.307,E2 -18200.307} C_VEL
LIN {X 0,Y 263.201,Z 180.699,A -85,B 0,C 180,E1 -18205.292,E2 -18205.292} C_VEL
LIN {X 0,Y 263.173,Z 180.693,A -85,B 0,C 180,E1 -18208.731,E2 -18208.731} C_VEL
LIN {X 0,Y 263.126,Z 180.696,A -85,B 0,C 180,E1 -18212.289,E2 -18212.289} C_VEL
LIN {X 0,Y 263.177,Z 180.663,A -85,B 0,C 180,E1 -18216.764,E2 -18216.764} C_VEL
LIN {X 0,Y 263.101,Z 180.714,A -85,B 0,C 180,E1 -18219.874,E2 -18219.874} C_VEL
LIN {X 0,Y 263.099,Z 180.677,A -85,B 0,C 180,E1 -18223.99,E2 -18223.99} C_VEL
LIN {X 0,Y 263.12,Z 180.698,A -85,B 0,C 180,E1 -18228.108,E2 -18228.108} C_VEL
LIN {X 0,Y 263.156,Z 180.694,A -85,B 0,C 180,E1 -18232.104,E2 -18232.104} C_VEL
LIN {X 0,Y 263.18,Z 180.84,A -85,B 0,C 180,E1 -18235.684,E2 -18235.684} C_VEL
LIN {X 0,Y 265.018,Z 188.428,A -85,B 0,C 180,E1 -18238.874,E2 -18238.874} C_VEL
LIN {X 0,Y 268.093,Z 195.155,A -85,B 0,C 180,E1 -18239.541,E2 -18239.541} C_VEL
LIN {X 0,Y 273.981,Z 208.412,A -85,B 0,C 180,E1 -18240.656,E2 -18240.656} C_VEL
LIN {X 0,Y 278.016,Z 219.111,A -85,B 0,C 180,E1 -18241.433,E2 -18241.433} C_VEL
LIN {X 0,Y 279.709,Z 229.535,A -85,B 0,C 180,E1 -18241.921,E2 -18241.921} C_VEL
LIN {X 0,Y 277.638,Z 296.55,A -85,B 0,C 180,E1 -18243.656,E2 -18243.656} C_VEL
LIN {X 0,Y 276.514,Z 310.279,A -85,B 0,C 180,E1 -18244.301,E2 -18244.301} C_VEL
LIN {X 0,Y 275.266,Z 322.604,A -85,B 0,C 180,E1 -18245.187,E2 -18245.187} C_VEL
LIN {X 0,Y 273.544,Z 334.429,A -85,B 0,C 180,E1 -18246.333,E2 -18246.333} C_VEL
LIN {X 0,Y 271.608,Z 345.789,A -85,B 0,C 180,E1 -18247.765,E2 -18247.765} C_VEL
LIN {X 0,Y 269.745,Z 356.027,A -85,B 0,C 180,E1 -18249.408,E2 -18249.408} C_VEL
LIN {X 0,Y 267.9,Z 365.536,A -85,B 0,C 180,E1 -18251.334,E2 -18251.334} C_VEL
LIN {X 0,Y 266.003,Z 374.148,A -85,B 0,C 180,E1 -18253.501,E2 -18253.501} C_VEL
LIN {X 0,Y 264.356,Z 381.339,A -85,B 0,C 180,E1 -18255.765,E2 -18255.765} C_VEL
LIN {X 0,Y 263.311,Z 386.188,A -85,B 0,C 180,E1 -18257.672,E2 -18257.672} C_VEL
LIN {X 0,Y 262.343,Z 390.902,A -85,B 0,C 180,E1 -18259.973,E2 -18259.973} C_VEL
LIN {X 0,Y 261.684,Z 394.509,A -85,B 0,C 180,E1 -18262.284,E2 -18262.284} C_VEL
LIN {X 0,Y 261.352,Z 396.783,A -85,B 0,C 180,E1 -18264.252,E2 -18264.252} C_VEL
LIN {X 0,Y 261.123,Z 398.771,A -85,B 0,C 180,E1 -18266.915,E2 -18266.915} C_VEL
LIN {X 0,Y 261.076,Z 399.615,A -85,B 0,C 180,E1 -18270.001,E2 -18270.001} C_VEL
LIN {X 0,Y 261.057,Z 399.421,A -85,B 0,C 180,E1 -18271.543,E2 -18271.543} C_VEL
LIN {X 0,Y 261.121,Z 398.832,A -85,B 0,C 180,E1 -18273.086,E2 -18273.086} C_VEL
LIN {X 0,Y 261.404,Z 396.495,A -85,B 0,C 180,E1 -18276.174,E2 -18276.174} C_VEL
LIN {X 0,Y 261.879,Z 393.613,A -85,B 0,C 180,E1 -18278.488,E2 -18278.488} C_VEL
LIN {X 0,Y 262.598,Z 389.707,A -85,B 0,C 180,E1 -18280.798,E2 -18280.798} C_VEL
LIN {X 0,Y 263.676,Z 384.668,A -85,B 0,C 180,E1 -18283.095,E2 -18283.095} C_VEL
LIN {X 0,Y 265.068,Z 378.325,A -85,B 0,C 180,E1 -18285.376,E2 -18285.376} C_VEL
LIN {X 0,Y 266.896,Z 370.389,A -85,B 0,C 180,E1 -18287.627,E2 -18287.627} C_VEL
LIN {X 0,Y 268.736,Z 361.314,A -85,B 0,C 180,E1 -18289.698,E2 -18289.698} C_VEL
LIN {X 0,Y 270.623,Z 351.334,A -85,B 0,C 180,E1 -18291.52,E2 -18291.52} C_VEL
LIN {X 0,Y 272.744,Z 339.902,A -85,B 0,C 180,E1 -18293.139,E2 -18293.139} C_VEL
LIN {X 0,Y 274.453,Z 328.677,A -85,B 0,C 180,E1 -18294.388,E2 -18294.388} C_VEL
LIN {X 0,Y 276.022,Z 316.014,A -85,B 0,C 180,E1 -18295.446,E2 -18295.446} C_VEL
LIN {X 0,Y 277.201,Z 303.313,A -85,B 0,C 180,E1 -18296.187,E2 -18296.187} C_VEL
LIN {X 0,Y 277.933,Z 290.211,A -85,B 0,C 180,E1 -18296.669,E2 -18296.669} C_VEL
LIN {X 0,Y 279.65,Z 228.132,A -85,B 0,C 180,E1 -18298.254,E2 -18298.254} C_VEL
LIN {X 0,Y 277.739,Z 217.967,A -85,B 0,C 180,E1 -18298.76,E2 -18298.76} C_VEL
LIN {X 0,Y 270.954,Z 201.265,A -85,B 0,C 180,E1 -18300.051,E2 -18300.051} C_VEL
LIN {X 0,Y 265.062,Z 188.481,A -85,B 0,C 180,E1 -18301.246,E2 -18301.246} C_VEL
LIN {X 0,Y 263.201,Z 180.838,A -85,B 0,C 180,E1 -18304.453,E2 -18304.453} C_VEL
LIN {X 0,Y 263.166,Z 180.696,A -85,B 0,C 180,E1 -18307.896,E2 -18307.896} C_VEL
LIN {X 0,Y 263.124,Z 180.694,A -85,B 0,C 180,E1 -18311.893,E2 -18311.893} C_VEL
LIN {X 0,Y 263.105,Z 180.676,A -85,B 0,C 180,E1 -18316.155,E2 -18316.155} C_VEL
LIN {X 0,Y 263.105,Z 180.712,A -85,B 0,C 180,E1 -18320.127,E2 -18320.127} C_VEL
LIN {X 0,Y 263.162,Z 180.656,A -85,B 0,C 180,E1 -18324.018,E2 -18324.018} C_VEL
LIN {X 0,Y 263.131,Z 180.693,A -85,B 0,C 180,E1 -18327.711,E2 -18327.711} C_VEL
LIN {X 0,Y 263.199,Z 180.687,A -85,B 0,C 180,E1 -18331.783,E2 -18331.783} C_VEL
LIN {X 0,Y 263.199,Z 180.7,A -85,B 0,C 180,E1 -18335.212,E2 -18335.212} C_VEL
LIN {X 0,Y 263.26,Z 180.685,A -85,B 0,C 180,E1 -18339.693,E2 -18339.693} C_VEL
LIN {X 0,Y 263.342,Z 180.662,A -85,B 0,C 180,E1 -18344.521,E2 -18344.521} C_VEL
LIN {X 0,Y 263.371,Z 180.667,A -85,B 0,C 180,E1 -18349.234,E2 -18349.234} C_VEL
LIN {X 0,Y 263.457,Z 180.646,A -85,B 0,C 180,E1 -18350.175,E2 -18350.175} C_VEL
LIN {X 0,Y 262.892,Z 180.718,A -85,B 0,C 180,E1 -18351.45,E2 -18351.45} C_VEL
LIN {X 0,Y 260.024,Z 181.092,A -85,B 0,C 180,E1 -18353.527,E2 -18353.527} C_VEL
LIN {X 0,Y 257.558,Z 181.399,A -85,B 0,C 180,E1 -18355.217,E2 -18355.217} C_VEL
LIN {X 0,Y 256.55,Z 181.512,A -85,B 0,C 180,E1 -18356.53,E2 -18356.53} C_VEL
LIN {X 0,Y 256.5,Z 181.515,A -85,B 0,C 180,E1 -18356.974,E2 -18356.974} C_VEL
LIN {X 0,Y 256.754,Z 181.499,A -85,B 0,C 180,E1 -18360,E2 -18360} C_VEL
LIN {X 0,Y 256.49,Z 181.523,A -85,B 0,C 180,E1 -18363.141,E2 -18363.141} C_VEL
LIN {X 0,Y 256.5,Z 181.534,A -85,B 0,C 180,E1 -18367.874,E2 -18367.874} C_VEL
LIN {X 0,Y 256.252,Z 181.553,A -85,B 0,C 180,E1 -18372.674,E2 -18372.674} C_VEL
LIN {X 0,Y 256.24,Z 181.56,A -85,B 0,C 180,E1 -18376.271,E2 -18376.271} C_VEL
LIN {X 0,Y 256.147,Z 181.579,A -85,B 0,C 180,E1 -18380.897,E2 -18380.897} C_VEL
LIN {X 0,Y 256.168,Z 181.565,A -85,B 0,C 180,E1 -18385.13,E2 -18385.13} C_VEL
LIN {X 0,Y 256.102,Z 181.571,A -85,B 0,C 180,E1 -18389.601,E2 -18389.601} C_VEL
LIN {X 0,Y 256.066,Z 181.581,A -85,B 0,C 180,E1 -18393.293,E2 -18393.293} C_VEL
LIN {X 0,Y 256.113,Z 181.536,A -85,B 0,C 180,E1 -18397.271,E2 -18397.271} C_VEL
LIN {X 0,Y 256.054,Z 181.589,A -85,B 0,C 180,E1 -18401.204,E2 -18401.204} C_VEL
LIN {X 0,Y 256.04,Z 181.591,A -85,B 0,C 180,E1 -18405.534,E2 -18405.534} C_VEL
LIN {X 0,Y 256.055,Z 181.592,A -85,B 0,C 180,E1 -18408.797,E2 -18408.797} C_VEL
LIN {X 0,Y 256.174,Z 181.76,A -85,B 0,C 180,E1 -18413.366,E2 -18413.366} C_VEL
LIN {X 0,Y 258.146,Z 190.033,A -85,B 0,C 180,E1 -18417.01,E2 -18417.01} C_VEL
LIN {X 0,Y 258.738,Z 192.641,A -85,B 0,C 180,E1 -18417.964,E2 -18417.964} C_VEL
LIN {X 0,Y 265.761,Z 208.244,A -85,B 0,C 180,E1 -18419.429,E2 -18419.429} C_VEL
LIN {X 0,Y 270.406,Z 219.751,A -85,B 0,C 180,E1 -18420.352,E2 -18420.352} C_VEL
LIN {X 0,Y 273.286,Z 237.338,A -85,B 0,C 180,E1 -18421.213,E2 -18421.213} C_VEL
LIN {X 0,Y 271.244,Z 300.589,A -85,B 0,C 180,E1 -18422.88,E2 -18422.88} C_VEL
LIN {X 0,Y 270.101,Z 314.481,A -85,B 0,C 180,E1 -18423.539,E2 -18423.539} C_VEL
LIN {X 0,Y 268.589,Z 326.908,A -85,B 0,C 180,E1 -18424.422,E2 -18424.422} C_VEL
LIN {X 0,Y 266.736,Z 339.577,A -85,B 0,C 180,E1 -18425.689,E2 -18425.689} C_VEL
LIN {X 0,Y 264.746,Z 350.838,A -85,B 0,C 180,E1 -18427.155,E2 -18427.155} C_VEL
LIN {X 0,Y 262.681,Z 360.981,A -85,B 0,C 180,E1 -18428.826,E2 -18428.826} C_VEL
LIN {X 0,Y 260.702,Z 370.618,A -85,B 0,C 180,E1 -18430.843,E2 -18430.843} C_VEL
LIN {X 0,Y 258.838,Z 379.017,A -85,B 0,C 180,E1 -18433.029,E2 -18433.029} C_VEL
LIN {X 0,Y 257.089,Z 386.175,A -85,B 0,C 180,E1 -18435.352,E2 -18435.352} C_VEL
LIN {X 0,Y 255.652,Z 392.694,A -85,B 0,C 180,E1 -18438.101,E2 -18438.101} C_VEL
LIN {X 0,Y 254.803,Z 397.006,A -85,B 0,C 180,E1 -18440.474,E2 -18440.474} C_VEL
LIN {X 0,Y 254.416,Z 399.29,A -85,B 0,C 180,E1 -18442.06,E2 -18442.06} C_VEL
LIN {X 0,Y 254.022,Z 402.264,A -85,B 0,C 180,E1 -18444.881,E2 -18444.881} C_VEL
LIN {X 0,Y 253.924,Z 403.513,A -85,B 0,C 180,E1 -18446.826,E2 -18446.826} C_VEL
LIN {X 0,Y 253.948,Z 404.116,A -85,B 0,C 180,E1 -18448.413,E2 -18448.413} C_VEL
LIN {X 0,Y 253.981,Z 404.327,A -85,B 0,C 180,E1 -18449.999,E2 -18449.999} C_VEL
LIN {X 0,Y 253.948,Z 404.106,A -85,B 0,C 180,E1 -18451.585,E2 -18451.585} C_VEL
LIN {X 0,Y 254.014,Z 402.503,A -85,B 0,C 180,E1 -18454.76,E2 -18454.76} C_VEL
LIN {X 0,Y 254.168,Z 401.107,A -85,B 0,C 180,E1 -18456.349,E2 -18456.349} C_VEL
LIN {X 0,Y 254.606,Z 398.178,A -85,B 0,C 180,E1 -18458.731,E2 -18458.731} C_VEL
LIN {X 0,Y 255.328,Z 394.213,A -85,B 0,C 180,E1 -18461.108,E2 -18461.108} C_VEL
LIN {X 0,Y 256.609,Z 388.115,A -85,B 0,C 180,E1 -18463.865,E2 -18463.865} C_VEL
LIN {X 0,Y 258.212,Z 381.454,A -85,B 0,C 180,E1 -18466.198,E2 -18466.198} C_VEL
LIN {X 0,Y 260.103,Z 373.188,A -85,B 0,C 180,E1 -18468.51,E2 -18468.51} C_VEL
LIN {X 0,Y 261.851,Z 364.706,A -85,B 0,C 180,E1 -18470.42,E2 -18470.42} C_VEL
LIN {X 0,Y 263.98,Z 354.226,A -85,B 0,C 180,E1 -18472.294,E2 -18472.294} C_VEL
LIN {X 0,Y 266.17,Z 342.424,A -85,B 0,C 180,E1 -18473.95,E2 -18473.95} C_VEL
LIN {X 0,Y 268.068,Z 330.533,A -85,B 0,C 180,E1 -18475.214,E2 -18475.214} C_VEL
LIN {X 0,Y 269.581,Z 318.151,A -85,B 0,C 180,E1 -18476.202,E2 -18476.202} C_VEL
LIN {X 0,Y 270.86,Z 305.393,A -85,B 0,C 180,E1 -18476.9,E2 -18476.9} C_VEL
LIN {X 0,Y 271.551,Z 291.89,A -85,B 0,C 180,E1 -18477.346,E2 -18477.346} C_VEL
LIN {X 0,Y 273.214,Z 237.384,A -85,B 0,C 180,E1 -18478.754,E2 -18478.754} C_VEL
LIN {X 0,Y 270.157,Z 219.143,A -85,B 0,C 180,E1 -18479.654,E2 -18479.654} C_VEL
LIN {X 0,Y 263.524,Z 203.102,A -85,B 0,C 180,E1 -18480.973,E2 -18480.973} C_VEL
LIN {X 0,Y 258.68,Z 192.532,A -85,B 0,C 180,E1 -18482.009,E2 -18482.009} C_VEL
LIN {X 0,Y 257.246,Z 186.22,A -85,B 0,C 180,E1 -18484.574,E2 -18484.574} C_VEL
LIN {X 0,Y 256.173,Z 181.623,A -85,B 0,C 180,E1 -18486.693,E2 -18486.693} C_VEL
LIN {X 0,Y 256.051,Z 181.592,A -85,B 0,C 180,E1 -18491.202,E2 -18491.202} C_VEL
LIN {X 0,Y 256.036,Z 181.588,A -85,B 0,C 180,E1 -18495.533,E2 -18495.533} C_VEL
LIN {X 0,Y 256.049,Z 181.59,A -85,B 0,C 180,E1 -18498.795,E2 -18498.795} C_VEL
LIN {X 0,Y 256.124,Z 181.533,A -85,B 0,C 180,E1 -18502.866,E2 -18502.866} C_VEL
LIN {X 0,Y 256.061,Z 181.582,A -85,B 0,C 180,E1 -18506.706,E2 -18506.706} C_VEL
LIN {X 0,Y 256.097,Z 181.571,A -85,B 0,C 180,E1 -18510.398,E2 -18510.398} C_VEL
LIN {X 0,Y 256.163,Z 181.565,A -85,B 0,C 180,E1 -18514.87,E2 -18514.87} C_VEL
LIN {X 0,Y 256.141,Z 181.579,A -85,B 0,C 180,E1 -18519.103,E2 -18519.103} C_VEL
LIN {X 0,Y 256.25,Z 181.561,A -85,B 0,C 180,E1 -18524.082,E2 -18524.082} C_VEL
LIN {X 0,Y 256.281,Z 181.549,A -85,B 0,C 180,E1 -18527.327,E2 -18527.327} C_VEL
LIN {X 0,Y 256.472,Z 181.531,A -85,B 0,C 180,E1 -18530.56,E2 -18530.56} C_VEL
LIN {X 0,Y 256.474,Z 181.528,A -85,B 0,C 180,E1 -18533.707,E2 -18533.707} C_VEL
LIN {X 0,Y 256.704,Z 181.509,A -85,B 0,C 180,E1 -18538.431,E2 -18538.431} C_VEL
LIN {X 0,Y 256.704,Z 181.49,A -85,B 0,C 180,E1 -18541.569,E2 -18541.569} C_VEL
LIN {X 0,Y 256.531,Z 181.516,A -85,B 0,C 180,E1 -18547.873,E2 -18547.873} C_VEL
LIN {X 0,Y 256.301,Z 181.55,A -85,B 0,C 180,E1 -18551.067,E2 -18551.067} C_VEL
LIN {X 0,Y 256.286,Z 181.54,A -85,B 0,C 180,E1 -18555.916,E2 -18555.916} C_VEL
LIN {X 0,Y 256.159,Z 181.566,A -85,B 0,C 180,E1 -18560.896,E2 -18560.896} C_VEL
LIN {X 0,Y 256.181,Z 181.574,A -85,B 0,C 180,E1 -18565.139,E2 -18565.139} C_VEL
LIN {X 0,Y 256.107,Z 181.58,A -85,B 0,C 180,E1 -18569.601,E2 -18569.601} C_VEL
LIN {X 0,Y 256.062,Z 181.554,A -85,B 0,C 180,E1 -18573.294,E2 -18573.294} C_VEL
LIN {X 0,Y 256.108,Z 181.551,A -85,B 0,C 180,E1 -18577.272,E2 -18577.272} C_VEL
LIN {X 0,Y 256.049,Z 181.576,A -85,B 0,C 180,E1 -18581.205,E2 -18581.205} C_VEL
LIN {X 0,Y 256.05,Z 181.574,A -85,B 0,C 180,E1 -18585.532,E2 -18585.532} C_VEL
LIN {X 0,Y 256.05,Z 181.567,A -85,B 0,C 180,E1 -18588.798,E2 -18588.798} C_VEL
LIN {X 0,Y 256.127,Z 181.583,A -85,B 0,C 180,E1 -18592.869,E2 -18592.869} C_VEL
LIN {X 0,Y 256.124,Z 181.606,A -85,B 0,C 180,E1 -18594.816,E2 -18594.816} C_VEL
LIN {X 0,Y 257.471,Z 187.316,A -85,B 0,C 180,E1 -18597.467,E2 -18597.467} C_VEL
LIN {X 0,Y 257.874,Z 188.854,A -85,B 0,C 180,E1 -18597.961,E2 -18597.961} C_VEL
LIN {X 0,Y 266.139,Z 206.422,A -85,B 0,C 180,E1 -18599.638,E2 -18599.638} C_VEL
LIN {X 0,Y 271.901,Z 220.907,A -85,B 0,C 180,E1 -18600.78,E2 -18600.78} C_VEL
LIN {X 0,Y 273.453,Z 230.252,A -85,B 0,C 180,E1 -18601.238,E2 -18601.238} C_VEL
LIN {X 0,Y 271.407,Z 295.482,A -85,B 0,C 180,E1 -18602.951,E2 -18602.951} C_VEL
LIN {X 0,Y 270.279,Z 308.832,A -85,B 0,C 180,E1 -18603.559,E2 -18603.559} C_VEL
LIN {X 0,Y 268.972,Z 321.585,A -85,B 0,C 180,E1 -18604.462,E2 -18604.462} C_VEL
LIN {X 0,Y 267.318,Z 332.914,A -85,B 0,C 180,E1 -18605.54,E2 -18605.54} C_VEL
LIN {X 0,Y 265.309,Z 344.569,A -85,B 0,C 180,E1 -18607.002,E2 -18607.002} C_VEL
LIN {X 0,Y 263.271,Z 355.037,A -85,B 0,C 180,E1 -18608.673,E2 -18608.673} C_VEL
LIN {X 0,Y 261.401,Z 364.576,A -85,B 0,C 180,E1 -18610.594,E2 -18610.594} C_VEL
LIN {X 0,Y 259.552,Z 372.863,A -85,B 0,C 180,E1 -18612.673,E2 -18612.673} C_VEL
